LIN {X 0,Y 421.046,Z 301.335,A -85,B 0,C 180,E1 -10144.338,E2 -10144.338} C_VEL
LIN {X 0,Y 421.385,Z 304.023,A -85,B 0,C 180,E1 -10144.837,E2 -10144.837} C_VEL
LIN {X 0,Y 420.511,Z 320.205,A -85,B 0,C 180,E1 -10147.657,E2 -10147.657} C_VEL
LIN {X 0,Y 419.69,Z 337.101,A -85,B 0,C 180,E1 -10150.579,E2 -10150.579} C_VEL
LIN {X 0,Y 422.949,Z 357.604,A -85,B 0,C 180,E1 -10151.184,E2 -10151.184} C_VEL
LIN {X 0,Y 424.065,Z 368.601,A -85,B 0,C 180,E1 -10151.466,E2 -10151.466} C_VEL
LIN {X 0,Y 422.703,Z 448.202,A -85,B 0,C 180,E1 -10153.026,E2 -10153.026} C_VEL
LIN {X 0,Y 422.076,Z 462.168,A -85,B 0,C 180,E1 -10153.498,E2 -10153.498} C_VEL
LIN {X 0,Y 421.349,Z 475.179,A -85,B 0,C 180,E1 -10154.153,E2 -10154.153} C_VEL
LIN {X 0,Y 420.586,Z 487.585,A -85,B 0,C 180,E1 -10154.992,E2 -10154.992} C_VEL
LIN {X 0,Y 419.764,Z 499.223,A -85,B 0,C 180,E1 -10156.002,E2 -10156.002} C_VEL
LIN {X 0,Y 419.009,Z 509.823,A -85,B 0,C 180,E1 -10157.162,E2 -10157.162} C_VEL
LIN {X 0,Y 418.449,Z 518.856,A -85,B 0,C 180,E1 -10158.375,E2 -10158.375} C_VEL
LIN {X 0,Y 417.83,Z 527.672,A -85,B 0,C 180,E1 -10159.83,E2 -10159.83} C_VEL
LIN {X 0,Y 417.483,Z 534.743,A -85,B 0,C 180,E1 -10161.288,E2 -10161.288} C_VEL
LIN {X 0,Y 417.25,Z 540.419,A -85,B 0,C 180,E1 -10162.745,E2 -10162.745} C_VEL
LIN {X 0,Y 417.115,Z 544.874,A -85,B 0,C 180,E1 -10164.2,E2 -10164.2} C_VEL
LIN {X 0,Y 417.146,Z 547.246,A -85,B 0,C 180,E1 -10165.17,E2 -10165.17} C_VEL
LIN {X 0,Y 417.051,Z 549.135,A -85,B 0,C 180,E1 -10166.137,E2 -10166.137} C_VEL
LIN {X 0,Y 417.124,Z 550.576,A -85,B 0,C 180,E1 -10167.105,E2 -10167.105} C_VEL
LIN {X 0,Y 417.122,Z 551.604,A -85,B 0,C 180,E1 -10168.071,E2 -10168.071} C_VEL
LIN {X 0,Y 417.096,Z 552.225,A -85,B 0,C 180,E1 -10169.036,E2 -10169.036} C_VEL
LIN {X 0,Y 417.123,Z 552.395,A -85,B 0,C 180,E1 -10170.002,E2 -10170.002} C_VEL
LIN {X 0,Y 417.109,Z 552.146,A -85,B 0,C 180,E1 -10170.967,E2 -10170.967} C_VEL
LIN {X 0,Y 417.123,Z 551.496,A -85,B 0,C 180,E1 -10171.932,E2 -10171.932} C_VEL
LIN {X 0,Y 417.156,Z 550.435,A -85,B 0,C 180,E1 -10172.898,E2 -10172.898} C_VEL
LIN {X 0,Y 417.054,Z 548.89,A -85,B 0,C 180,E1 -10173.866,E2 -10173.866} C_VEL
LIN {X 0,Y 417.143,Z 545.765,A -85,B 0,C 180,E1 -10175.318,E2 -10175.318} C_VEL
LIN {X 0,Y 417.233,Z 541.533,A -85,B 0,C 180,E1 -10176.772,E2 -10176.772} C_VEL
LIN {X 0,Y 417.443,Z 535.054,A -85,B 0,C 180,E1 -10178.472,E2 -10178.472} C_VEL
LIN {X 0,Y 417.739,Z 527.969,A -85,B 0,C 180,E1 -10179.931,E2 -10179.931} C_VEL
LIN {X 0,Y 418.276,Z 519.076,A -85,B 0,C 180,E1 -10181.387,E2 -10181.387} C_VEL
LIN {X 0,Y 418.823,Z 509.96,A -85,B 0,C 180,E1 -10182.6,E2 -10182.6} C_VEL
LIN {X 0,Y 419.403,Z 499.932,A -85,B 0,C 180,E1 -10183.692,E2 -10183.692} C_VEL
LIN {X 0,Y 420.108,Z 488.819,A -85,B 0,C 180,E1 -10184.657,E2 -10184.657} C_VEL
LIN {X 0,Y 420.808,Z 476.413,A -85,B 0,C 180,E1 -10185.499,E2 -10185.499} C_VEL
LIN {X 0,Y 421.393,Z 464.719,A -85,B 0,C 180,E1 -10186.097,E2 -10186.097} C_VEL
LIN {X 0,Y 421.903,Z 452.292,A -85,B 0,C 180,E1 -10186.543,E2 -10186.543} C_VEL
LIN {X 0,Y 422.237,Z 433.946,A -85,B 0,C 180,E1 -10186.935,E2 -10186.935} C_VEL
LIN {X 0,Y 423.043,Z 365.545,A -85,B 0,C 180,E1 -10188.216,E2 -10188.216} C_VEL
LIN {X 0,Y 419.504,Z 339.754,A -85,B 0,C 180,E1 -10188.877,E2 -10188.877} C_VEL
LIN {X 0,Y 420.603,Z 320.904,A -85,B 0,C 180,E1 -10192.341,E2 -10192.341} C_VEL
LIN {X 0,Y 421.565,Z 304.734,A -85,B 0,C 180,E1 -10195.354,E2 -10195.354} C_VEL
LIN {X 0,Y 418.666,Z 290.263,A -85,B 0,C 180,E1 -10198.307,E2 -10198.307} C_VEL
LIN {X 0,Y 418.272,Z 288.385,A -85,B 0,C 180,E1 -10198.733,E2 -10198.733} C_VEL
LIN {X 0,Y 418.205,Z 288.39,A -85,B 0,C 180,E1 -10201.395,E2 -10201.395} C_VEL
LIN {X 0,Y 418.246,Z 288.389,A -85,B 0,C 180,E1 -10204.576,E2 -10204.576} C_VEL
LIN {X 0,Y 418.209,Z 288.388,A -85,B 0,C 180,E1 -10207.829,E2 -10207.829} C_VEL
LIN {X 0,Y 418.197,Z 288.393,A -85,B 0,C 180,E1 -10210.948,E2 -10210.948} C_VEL
LIN {X 0,Y 418.19,Z 288.39,A -85,B 0,C 180,E1 -10213.726,E2 -10213.726} C_VEL
LIN {X 0,Y 418.186,Z 288.393,A -85,B 0,C 180,E1 -10216.445,E2 -10216.445} C_VEL
LIN {X 0,Y 418.192,Z 288.393,A -85,B 0,C 180,E1 -10219.131,E2 -10219.131} C_VEL
LIN {X 0,Y 418.217,Z 288.393,A -85,B 0,C 180,E1 -10222.773,E2 -10222.773} C_VEL
LIN {X 0,Y 418.211,Z 288.389,A -85,B 0,C 180,E1 -10226.319,E2 -10226.319} C_VEL
LIN {X 0,Y 418.22,Z 288.388,A -85,B 0,C 180,E1 -10229.725,E2 -10229.725} C_VEL
LIN {X 0,Y 418.239,Z 288.389,A -85,B 0,C 180,E1 -10233.018,E2 -10233.018} C_VEL
LIN {X 0,Y 418.24,Z 288.385,A -85,B 0,C 180,E1 -10236.216,E2 -10236.216} C_VEL
LIN {X 0,Y 418.22,Z 288.389,A -85,B 0,C 180,E1 -10239.335,E2 -10239.335} C_VEL
LIN {X 0,Y 418.249,Z 288.384,A -85,B 0,C 180,E1 -10242.394,E2 -10242.394} C_VEL
LIN {X 0,Y 418.27,Z 288.383,A -85,B 0,C 180,E1 -10245.401,E2 -10245.401} C_VEL
LIN {X 0,Y 418.291,Z 288.379,A -85,B 0,C 180,E1 -10248.368,E2 -10248.368} C_VEL
LIN {X 0,Y 418.484,Z 288.355,A -85,B 0,C 180,E1 -10252.278,E2 -10252.278} C_VEL
LIN {X 0,Y 418.474,Z 288.357,A -85,B 0,C 180,E1 -10254.216,E2 -10254.216} C_VEL
LIN {X 0,Y 418.508,Z 288.354,A -85,B 0,C 180,E1 -10258.075,E2 -10258.075} C_VEL
LIN {X 0,Y 418.636,Z 288.337,A -85,B 0,C 180,E1 -10260,E2 -10260} C_VEL
LIN {X 0,Y 418.466,Z 288.359,A -85,B 0,C 180,E1 -10262.888,E2 -10262.888} C_VEL
LIN {X 0,Y 418.456,Z 288.36,A -85,B 0,C 180,E1 -10266.751,E2 -10266.751} C_VEL
LIN {X 0,Y 418.313,Z 288.378,A -85,B 0,C 180,E1 -10269.672,E2 -10269.672} C_VEL
LIN {X 0,Y 418.325,Z 288.377,A -85,B 0,C 180,E1 -10273.006,E2 -10273.006} C_VEL
LIN {X 0,Y 418.282,Z 288.381,A -85,B 0,C 180,E1 -10276.735,E2 -10276.735} C_VEL
LIN {X 0,Y 418.24,Z 288.387,A -85,B 0,C 180,E1 -10279.79,E2 -10279.79} C_VEL
LIN {X 0,Y 418.21,Z 288.39,A -85,B 0,C 180,E1 -10282.737,E2 -10282.737} C_VEL
LIN {X 0,Y 418.243,Z 288.386,A -85,B 0,C 180,E1 -10285.905,E2 -10285.905} C_VEL
LIN {X 0,Y 418.248,Z 288.386,A -85,B 0,C 180,E1 -10289.163,E2 -10289.163} C_VEL
LIN {X 0,Y 418.234,Z 288.387,A -85,B 0,C 180,E1 -10292.845,E2 -10292.845} C_VEL
LIN {X 0,Y 418.226,Z 288.389,A -85,B 0,C 180,E1 -10296.24,E2 -10296.24} C_VEL
LIN {X 0,Y 418.245,Z 288.387,A -85,B 0,C 180,E1 -10299.682,E2 -10299.682} C_VEL
LIN {X 0,Y 418.227,Z 288.39,A -85,B 0,C 180,E1 -10302.325,E2 -10302.325} C_VEL
LIN {X 0,Y 418.233,Z 288.387,A -85,B 0,C 180,E1 -10305.112,E2 -10305.112} C_VEL
LIN {X 0,Y 418.277,Z 288.382,A -85,B 0,C 180,E1 -10307.775,E2 -10307.775} C_VEL
LIN {X 0,Y 418.254,Z 288.386,A -85,B 0,C 180,E1 -10311.561,E2 -10311.561} C_VEL
LIN {X 0,Y 418.249,Z 288.385,A -85,B 0,C 180,E1 -10315.16,E2 -10315.16} C_VEL
LIN {X 0,Y 418.235,Z 288.387,A -85,B 0,C 180,E1 -10317.473,E2 -10317.473} C_VEL
LIN {X 0,Y 418.261,Z 288.385,A -85,B 0,C 180,E1 -10320.896,E2 -10320.896} C_VEL
LIN {X 0,Y 418.264,Z 288.384,A -85,B 0,C 180,E1 -10324.097,E2 -10324.097} C_VEL
LIN {X 0,Y 418.233,Z 288.387,A -85,B 0,C 180,E1 -10327.264,E2 -10327.264} C_VEL
LIN {X 0,Y 418.279,Z 288.382,A -85,B 0,C 180,E1 -10330.364,E2 -10330.364} C_VEL
LIN {X 0,Y 418.314,Z 288.377,A -85,B 0,C 180,E1 -10333.405,E2 -10333.405} C_VEL
LIN {X 0,Y 418.343,Z 288.375,A -85,B 0,C 180,E1 -10336.999,E2 -10336.999} C_VEL
LIN {X 0,Y 418.339,Z 288.374,A -85,B 0,C 180,E1 -10340.328,E2 -10340.328} C_VEL
LIN {X 0,Y 418.511,Z 288.353,A -85,B 0,C 180,E1 -10342.279,E2 -10342.279} C_VEL
LIN {X 0,Y 418.511,Z 288.352,A -85,B 0,C 180,E1 -10344.216,E2 -10344.216} C_VEL
LIN {X 0,Y 418.542,Z 288.348,A -85,B 0,C 180,E1 -10348.074,E2 -10348.074} C_VEL
LIN {X 0,Y 418.67,Z 288.332,A -85,B 0,C 180,E1 -10349.998,E2 -10349.998} C_VEL
LIN {X 0,Y 418.507,Z 288.357,A -85,B 0,C 180,E1 -10352.886,E2 -10352.886} C_VEL
LIN {X 0,Y 418.482,Z 288.358,A -85,B 0,C 180,E1 -10356.749,E2 -10356.749} C_VEL
LIN {X 0,Y 418.352,Z 288.371,A -85,B 0,C 180,E1 -10359.17,E2 -10359.17} C_VEL
LIN {X 0,Y 418.363,Z 288.371,A -85,B 0,C 180,E1 -10362.611,E2 -10362.611} C_VEL
LIN {X 0,Y 418.324,Z 288.376,A -85,B 0,C 180,E1 -10363.36,E2 -10363.36} C_VEL
LIN {X 0,Y 417.633,Z 288.461,A -85,B 0,C 180,E1 -10364.163,E2 -10364.163} C_VEL
LIN {X 0,Y 414.749,Z 288.82,A -85,B 0,C 180,E1 -10365.468,E2 -10365.468} C_VEL
LIN {X 0,Y 412.33,Z 289.122,A -85,B 0,C 180,E1 -10366.522,E2 -10366.522} C_VEL
LIN {X 0,Y 411.306,Z 289.25,A -85,B 0,C 180,E1 -10367.337,E2 -10367.337} C_VEL
LIN {X 0,Y 411.23,Z 289.257,A -85,B 0,C 180,E1 -10367.613,E2 -10367.613} C_VEL
LIN {X 0,Y 411.221,Z 289.265,A -85,B 0,C 180,E1 -10371.029,E2 -10371.029} C_VEL
LIN {X 0,Y 411.214,Z 289.26,A -85,B 0,C 180,E1 -10374.212,E2 -10374.212} C_VEL
LIN {X 0,Y 411.243,Z 289.258,A -85,B 0,C 180,E1 -10377.474,E2 -10377.474} C_VEL
LIN {X 0,Y 411.182,Z 289.266,A -85,B 0,C 180,E1 -10380.843,E2 -10380.843} C_VEL
LIN {X 0,Y 411.183,Z 289.263,A -85,B 0,C 180,E1 -10384.33,E2 -10384.33} C_VEL
LIN {X 0,Y 411.179,Z 289.264,A -85,B 0,C 180,E1 -10387.969,E2 -10387.969} C_VEL
LIN {X 0,Y 411.255,Z 289.359,A -85,B 0,C 180,E1 -10391.508,E2 -10391.508} C_VEL
LIN {X 0,Y 412.397,Z 295.233,A -85,B 0,C 180,E1 -10392.933,E2 -10392.933} C_VEL
LIN {X 0,Y 414.802,Z 304.457,A -85,B 0,C 180,E1 -10393.227,E2 -10393.227} C_VEL
LIN {X 0,Y 416.781,Z 315.123,A -85,B 0,C 180,E1 -10393.524,E2 -10393.524} C_VEL
LIN {X 0,Y 415.341,Z 403.223,A -85,B 0,C 180,E1 -10395.224,E2 -10395.224} C_VEL
LIN {X 0,Y 415.04,Z 416.613,A -85,B 0,C 180,E1 -10395.683,E2 -10395.683} C_VEL
LIN {X 0,Y 414.55,Z 428.862,A -85,B 0,C 180,E1 -10396.29,E2 -10396.29} C_VEL
LIN {X 0,Y 413.945,Z 441.31,A -85,B 0,C 180,E1 -10397.127,E2 -10397.127} C_VEL
LIN {X 0,Y 413.301,Z 452.924,A -85,B 0,C 180,E1 -10398.132,E2 -10398.132} C_VEL
LIN {X 0,Y 412.687,Z 462.758,A -85,B 0,C 180,E1 -10399.193,E2 -10399.193} C_VEL
LIN {X 0,Y 412.002,Z 473.088,A -85,B 0,C 180,E1 -10400.583,E2 -10400.583} C_VEL
LIN {X 0,Y 411.43,Z 481.862,A -85,B 0,C 180,E1 -10402.053,E2 -10402.053} C_VEL
LIN {X 0,Y 410.983,Z 488.662,A -85,B 0,C 180,E1 -10403.476,E2 -10403.476} C_VEL
LIN {X 0,Y 410.578,Z 495.276,A -85,B 0,C 180,E1 -10405.237,E2 -10405.237} C_VEL
LIN {X 0,Y 410.367,Z 499.644,A -85,B 0,C 180,E1 -10406.768,E2 -10406.768} C_VEL
LIN {X 0,Y 410.18,Z 502.139,A -85,B 0,C 180,E1 -10407.917,E2 -10407.917} C_VEL
LIN {X 0,Y 410.024,Z 504.05,A -85,B 0,C 180,E1 -10409.056,E2 -10409.056} C_VEL
LIN {X 0,Y 409.943,Z 505.913,A -85,B 0,C 180,E1 -10410.953,E2 -10410.953} C_VEL
LIN {X 0,Y 409.95,Z 506.241,A -85,B 0,C 180,E1 -10413.043,E2 -10413.043} C_VEL
LIN {X 0,Y 410.043,Z 505.234,A -85,B 0,C 180,E1 -10414.629,E2 -10414.629} C_VEL
LIN {X 0,Y 410.195,Z 503.889,A -85,B 0,C 180,E1 -10415.72,E2 -10415.72} C_VEL
LIN {X 0,Y 410.366,Z 502.082,A -85,B 0,C 180,E1 -10416.803,E2 -10416.803} C_VEL
LIN {X 0,Y 410.635,Z 498.359,A -85,B 0,C 180,E1 -10418.41,E2 -10418.41} C_VEL
LIN {X 0,Y 411.045,Z 493.008,A -85,B 0,C 180,E1 -10420.095,E2 -10420.095} C_VEL
LIN {X 0,Y 411.519,Z 486.934,A -85,B 0,C 180,E1 -10421.583,E2 -10421.583} C_VEL
LIN {X 0,Y 412.174,Z 478.896,A -85,B 0,C 180,E1 -10423.15,E2 -10423.15} C_VEL
LIN {X 0,Y 412.849,Z 470.57,A -85,B 0,C 180,E1 -10424.448,E2 -10424.448} C_VEL
LIN {X 0,Y 413.65,Z 460.35,A -85,B 0,C 180,E1 -10425.74,E2 -10425.74} C_VEL
LIN {X 0,Y 414.424,Z 450.265,A -85,B 0,C 180,E1 -10426.766,E2 -10426.766} C_VEL
LIN {X 0,Y 415.041,Z 439.361,A -85,B 0,C 180,E1 -10427.656,E2 -10427.656} C_VEL
LIN {X 0,Y 415.674,Z 427.031,A -85,B 0,C 180,E1 -10428.435,E2 -10428.435} C_VEL
LIN {X 0,Y 416.13,Z 414.173,A -85,B 0,C 180,E1 -10429.032,E2 -10429.032} C_VEL
LIN {X 0,Y 416.469,Z 401.016,A -85,B 0,C 180,E1 -10429.426,E2 -10429.426} C_VEL
LIN {X 0,Y 418.135,Z 314.185,A -85,B 0,C 180,E1 -10431.159,E2 -10431.159} C_VEL
LIN {X 0,Y 415.58,Z 302.673,A -85,B 0,C 180,E1 -10431.56,E2 -10431.56} C_VEL
LIN {X 0,Y 412.825,Z 295.614,A -85,B 0,C 180,E1 -10431.896,E2 -10431.896} C_VEL
LIN {X 0,Y 411.408,Z 289.242,A -85,B 0,C 180,E1 -10433.194,E2 -10433.194} C_VEL
LIN {X 0,Y 411.417,Z 289.242,A -85,B 0,C 180,E1 -10437.063,E2 -10437.063} C_VEL
LIN {X 0,Y 411.586,Z 289.215,A -85,B 0,C 180,E1 -10440,E2 -10440} C_VEL
LIN {X 0,Y 411.417,Z 289.238,A -85,B 0,C 180,E1 -10442.938,E2 -10442.938} C_VEL
LIN {X 0,Y 411.404,Z 289.24,A -85,B 0,C 180,E1 -10446.868,E2 -10446.868} C_VEL
LIN {X 0,Y 411.246,Z 289.256,A -85,B 0,C 180,E1 -10449.84,E2 -10449.84} C_VEL
LIN {X 0,Y 411.264,Z 289.256,A -85,B 0,C 180,E1 -10453.11,E2 -10453.11} C_VEL
LIN {X 0,Y 411.21,Z 289.264,A -85,B 0,C 180,E1 -10456.891,E2 -10456.891} C_VEL
LIN {X 0,Y 411.163,Z 289.263,A -85,B 0,C 180,E1 -10459.991,E2 -10459.991} C_VEL
LIN {X 0,Y 411.157,Z 289.267,A -85,B 0,C 180,E1 -10463.151,E2 -10463.151} C_VEL
LIN {X 0,Y 411.195,Z 289.259,A -85,B 0,C 180,E1 -10466.384,E2 -10466.384} C_VEL
LIN {X 0,Y 411.16,Z 289.268,A -85,B 0,C 180,E1 -10469.716,E2 -10469.716} C_VEL
LIN {X 0,Y 411.169,Z 289.271,A -85,B 0,C 180,E1 -10473.16,E2 -10473.16} C_VEL
LIN {X 0,Y 411.16,Z 289.267,A -85,B 0,C 180,E1 -10476.557,E2 -10476.557} C_VEL
LIN {X 0,Y 411.195,Z 289.262,A -85,B 0,C 180,E1 -10479.734,E2 -10479.734} C_VEL
LIN {X 0,Y 411.148,Z 289.271,A -85,B 0,C 180,E1 -10483.137,E2 -10483.137} C_VEL
LIN {X 0,Y 411.141,Z 289.27,A -85,B 0,C 180,E1 -10485.886,E2 -10485.886} C_VEL
LIN {X 0,Y 411.139,Z 289.271,A -85,B 0,C 180,E1 -10488.776,E2 -10488.776} C_VEL
LIN {X 0,Y 411.168,Z 289.267,A -85,B 0,C 180,E1 -10492.03,E2 -10492.03} C_VEL
LIN {X 0,Y 411.188,Z 289.272,A -85,B 0,C 180,E1 -10495.671,E2 -10495.671} C_VEL
LIN {X 0,Y 411.174,Z 289.277,A -85,B 0,C 180,E1 -10499.156,E2 -10499.156} C_VEL
LIN {X 0,Y 411.242,Z 289.392,A -85,B 0,C 180,E1 -10501.493,E2 -10501.493} C_VEL
LIN {X 0,Y 414.104,Z 302.418,A -85,B 0,C 180,E1 -10504.092,E2 -10504.092} C_VEL
LIN {X 0,Y 414.521,Z 305.674,A -85,B 0,C 180,E1 -10504.715,E2 -10504.715} C_VEL
LIN {X 0,Y 413.497,Z 322.95,A -85,B 0,C 180,E1 -10507.784,E2 -10507.784} C_VEL
LIN {X 0,Y 412.843,Z 336.588,A -85,B 0,C 180,E1 -10510.177,E2 -10510.177} C_VEL
LIN {X 0,Y 416.359,Z 358.576,A -85,B 0,C 180,E1 -10510.855,E2 -10510.855} C_VEL
LIN {X 0,Y 417.425,Z 369.282,A -85,B 0,C 180,E1 -10511.137,E2 -10511.137} C_VEL
LIN {X 0,Y 415.99,Z 447.96,A -85,B 0,C 180,E1 -10512.712,E2 -10512.712} C_VEL
LIN {X 0,Y 415.37,Z 461.098,A -85,B 0,C 180,E1 -10513.16,E2 -10513.16} C_VEL
LIN {X 0,Y 414.685,Z 473.298,A -85,B 0,C 180,E1 -10513.765,E2 -10513.765} C_VEL
LIN {X 0,Y 413.791,Z 485.957,A -85,B 0,C 180,E1 -10514.614,E2 -10514.614} C_VEL
LIN {X 0,Y 412.985,Z 497.705,A -85,B 0,C 180,E1 -10515.629,E2 -10515.629} C_VEL
LIN {X 0,Y 412.225,Z 507.992,A -85,B 0,C 180,E1 -10516.746,E2 -10516.746} C_VEL
LIN {X 0,Y 411.465,Z 518.593,A -85,B 0,C 180,E1 -10518.175,E2 -10518.175} C_VEL
LIN {X 0,Y 410.8,Z 527.377,A -85,B 0,C 180,E1 -10519.654,E2 -10519.654} C_VEL
LIN {X 0,Y 410.427,Z 534.434,A -85,B 0,C 180,E1 -10521.137,E2 -10521.137} C_VEL
LIN {X 0,Y 410.17,Z 540.096,A -85,B 0,C 180,E1 -10522.619,E2 -10522.619} C_VEL
LIN {X 0,Y 410.036,Z 544.536,A -85,B 0,C 180,E1 -10524.099,E2 -10524.099} C_VEL
LIN {X 0,Y 410.053,Z 546.905,A -85,B 0,C 180,E1 -10525.086,E2 -10525.086} C_VEL
LIN {X 0,Y 409.968,Z 548.774,A -85,B 0,C 180,E1 -10526.07,E2 -10526.07} C_VEL
LIN {X 0,Y 410.022,Z 550.205,A -85,B 0,C 180,E1 -10527.054,E2 -10527.054} C_VEL
LIN {X 0,Y 410.048,Z 551.226,A -85,B 0,C 180,E1 -10528.037,E2 -10528.037} C_VEL
LIN {X 0,Y 410.016,Z 551.834,A -85,B 0,C 180,E1 -10529.02,E2 -10529.02} C_VEL
LIN {X 0,Y 410.039,Z 551.988,A -85,B 0,C 180,E1 -10530.002,E2 -10530.002} C_VEL
LIN {X 0,Y 410.028,Z 551.73,A -85,B 0,C 180,E1 -10530.984,E2 -10530.984} C_VEL
LIN {X 0,Y 410.051,Z 551.071,A -85,B 0,C 180,E1 -10531.966,E2 -10531.966} C_VEL
LIN {X 0,Y 410.054,Z 549.99,A -85,B 0,C 180,E1 -10532.949,E2 -10532.949} C_VEL
LIN {X 0,Y 409.97,Z 548.429,A -85,B 0,C 180,E1 -10533.933,E2 -10533.933} C_VEL
LIN {X 0,Y 410.059,Z 545.275,A -85,B 0,C 180,E1 -10535.41,E2 -10535.41} C_VEL
LIN {X 0,Y 410.165,Z 541.011,A -85,B 0,C 180,E1 -10536.89,E2 -10536.89} C_VEL
LIN {X 0,Y 410.363,Z 534.489,A -85,B 0,C 180,E1 -10538.619,E2 -10538.619} C_VEL
LIN {X 0,Y 410.693,Z 527.341,A -85,B 0,C 180,E1 -10540.103,E2 -10540.103} C_VEL
LIN {X 0,Y 411.273,Z 518.382,A -85,B 0,C 180,E1 -10541.583,E2 -10541.583} C_VEL
LIN {X 0,Y 411.876,Z 509.197,A -85,B 0,C 180,E1 -10542.816,E2 -10542.816} C_VEL
LIN {X 0,Y 412.474,Z 499.048,A -85,B 0,C 180,E1 -10543.926,E2 -10543.926} C_VEL
LIN {X 0,Y 413.198,Z 487.791,A -85,B 0,C 180,E1 -10544.907,E2 -10544.907} C_VEL
LIN {X 0,Y 413.941,Z 475.22,A -85,B 0,C 180,E1 -10545.763,E2 -10545.763} C_VEL
LIN {X 0,Y 414.535,Z 463.156,A -85,B 0,C 180,E1 -10546.371,E2 -10546.371} C_VEL
LIN {X 0,Y 415.081,Z 449.036,A -85,B 0,C 180,E1 -10546.855,E2 -10546.855} C_VEL
LIN {X 0,Y 415.934,Z 395.669,A -85,B 0,C 180,E1 -10547.89,E2 -10547.89} C_VEL
LIN {X 0,Y 416.24,Z 366.622,A -85,B 0,C 180,E1 -10548.454,E2 -10548.454} C_VEL
LIN {X 0,Y 412.547,Z 339.36,A -85,B 0,C 180,E1 -10549.175,E2 -10549.175} C_VEL
LIN {X 0,Y 413.717,Z 320.343,A -85,B 0,C 180,E1 -10552.734,E2 -10552.734} C_VEL
LIN {X 0,Y 414.634,Z 306.778,A -85,B 0,C 180,E1 -10555.305,E2 -10555.305} C_VEL
LIN {X 0,Y 412.16,Z 293.628,A -85,B 0,C 180,E1 -10558.014,E2 -10558.014} C_VEL
LIN {X 0,Y 411.234,Z 289.261,A -85,B 0,C 180,E1 -10558.948,E2 -10558.948} C_VEL
LIN {X 0,Y 411.159,Z 289.269,A -85,B 0,C 180,E1 -10561.996,E2 -10561.996} C_VEL
LIN {X 0,Y 411.196,Z 289.266,A -85,B 0,C 180,E1 -10564.875,E2 -10564.875} C_VEL
LIN {X 0,Y 411.183,Z 289.264,A -85,B 0,C 180,E1 -10568.164,E2 -10568.164} C_VEL
LIN {X 0,Y 411.15,Z 289.267,A -85,B 0,C 180,E1 -10571.806,E2 -10571.806} C_VEL
LIN {X 0,Y 411.16,Z 289.267,A -85,B 0,C 180,E1 -10575.507,E2 -10575.507} C_VEL
LIN {X 0,Y 411.133,Z 289.275,A -85,B 0,C 180,E1 -10578.772,E2 -10578.772} C_VEL
LIN {X 0,Y 411.166,Z 289.266,A -85,B 0,C 180,E1 -10582.023,E2 -10582.023} C_VEL
LIN {X 0,Y 411.183,Z 289.267,A -85,B 0,C 180,E1 -10585.122,E2 -10585.122} C_VEL
LIN {X 0,Y 411.14,Z 289.269,A -85,B 0,C 180,E1 -10588,E2 -10588} C_VEL
LIN {X 0,Y 411.191,Z 289.264,A -85,B 0,C 180,E1 -10591.407,E2 -10591.407} C_VEL
LIN {X 0,Y 411.19,Z 289.268,A -85,B 0,C 180,E1 -10594.932,E2 -10594.932} C_VEL
LIN {X 0,Y 411.176,Z 289.266,A -85,B 0,C 180,E1 -10597.911,E2 -10597.911} C_VEL
LIN {X 0,Y 411.19,Z 289.268,A -85,B 0,C 180,E1 -10601.049,E2 -10601.049} C_VEL
LIN {X 0,Y 411.226,Z 289.259,A -85,B 0,C 180,E1 -10604.13,E2 -10604.13} C_VEL
LIN {X 0,Y 411.275,Z 289.257,A -85,B 0,C 180,E1 -10607.164,E2 -10607.164} C_VEL
LIN {X 0,Y 411.264,Z 289.255,A -85,B 0,C 180,E1 -10610.16,E2 -10610.16} C_VEL
LIN {X 0,Y 411.425,Z 289.239,A -85,B 0,C 180,E1 -10613.132,E2 -10613.132} C_VEL
LIN {X 0,Y 411.273,Z 289.257,A -85,B 0,C 180,E1 -10615.098,E2 -10615.098} C_VEL
LIN {X 0,Y 411.477,Z 289.229,A -85,B 0,C 180,E1 -10618.042,E2 -10618.042} C_VEL
LIN {X 0,Y 411.606,Z 289.213,A -85,B 0,C 180,E1 -10620,E2 -10620} C_VEL
LIN {X 0,Y 411.423,Z 289.237,A -85,B 0,C 180,E1 -10622.937,E2 -10622.937} C_VEL
LIN {X 0,Y 411.42,Z 289.236,A -85,B 0,C 180,E1 -10626.867,E2 -10626.867} C_VEL
LIN {X 0,Y 411.266,Z 289.256,A -85,B 0,C 180,E1 -10629.839,E2 -10629.839} C_VEL
LIN {X 0,Y 411.283,Z 289.254,A -85,B 0,C 180,E1 -10633.108,E2 -10633.108} C_VEL
LIN {X 0,Y 411.229,Z 289.26,A -85,B 0,C 180,E1 -10636.889,E2 -10636.889} C_VEL
LIN {X 0,Y 411.182,Z 289.266,A -85,B 0,C 180,E1 -10639.989,E2 -10639.989} C_VEL
LIN {X 0,Y 411.175,Z 289.267,A -85,B 0,C 180,E1 -10643.149,E2 -10643.149} C_VEL
LIN {X 0,Y 411.212,Z 289.263,A -85,B 0,C 180,E1 -10646.382,E2 -10646.382} C_VEL
LIN {X 0,Y 411.185,Z 289.266,A -85,B 0,C 180,E1 -10649.713,E2 -10649.713} C_VEL
LIN {X 0,Y 411.184,Z 289.266,A -85,B 0,C 180,E1 -10653.157,E2 -10653.157} C_VEL
LIN {X 0,Y 411.174,Z 289.268,A -85,B 0,C 180,E1 -10656.554,E2 -10656.554} C_VEL
LIN {X 0,Y 411.208,Z 289.263,A -85,B 0,C 180,E1 -10659.731,E2 -10659.731} C_VEL
LIN {X 0,Y 411.16,Z 289.268,A -85,B 0,C 180,E1 -10663.135,E2 -10663.135} C_VEL
LIN {X 0,Y 411.205,Z 289.263,A -85,B 0,C 180,E1 -10665.875,E2 -10665.875} C_VEL
LIN {X 0,Y 411.196,Z 289.265,A -85,B 0,C 180,E1 -10668.766,E2 -10668.766} C_VEL
LIN {X 0,Y 411.192,Z 289.265,A -85,B 0,C 180,E1 -10672.029,E2 -10672.029} C_VEL
LIN {X 0,Y 411.196,Z 289.265,A -85,B 0,C 180,E1 -10675.668,E2 -10675.668} C_VEL
LIN {X 0,Y 411.18,Z 289.265,A -85,B 0,C 180,E1 -10679.153,E2 -10679.153} C_VEL
LIN {X 0,Y 411.252,Z 289.259,A -85,B 0,C 180,E1 -10682.523,E2 -10682.523} C_VEL
LIN {X 0,Y 411.221,Z 289.261,A -85,B 0,C 180,E1 -10685.785,E2 -10685.785} C_VEL
LIN {X 0,Y 411.192,Z 289.265,A -85,B 0,C 180,E1 -10688.966,E2 -10688.966} C_VEL
LIN {X 0,Y 411.249,Z 289.257,A -85,B 0,C 180,E1 -10692.085,E2 -10692.085} C_VEL
LIN {X 0,Y 411.257,Z 289.256,A -85,B 0,C 180,E1 -10695.147,E2 -10695.147} C_VEL
LIN {X 0,Y 411.281,Z 289.253,A -85,B 0,C 180,E1 -10698.167,E2 -10698.167} C_VEL
LIN {X 0,Y 411.48,Z 289.228,A -85,B 0,C 180,E1 -10702.146,E2 -10702.146} C_VEL
LIN {X 0,Y 411.473,Z 289.229,A -85,B 0,C 180,E1 -10704.117,E2 -10704.117} C_VEL
LIN {X 0,Y 411.511,Z 289.224,A -85,B 0,C 180,E1 -10708.041,E2 -10708.041} C_VEL
LIN {X 0,Y 411.639,Z 289.208,A -85,B 0,C 180,E1 -10709.998,E2 -10709.998} C_VEL
LIN {X 0,Y 411.463,Z 289.234,A -85,B 0,C 180,E1 -10712.935,E2 -10712.935} C_VEL
LIN {X 0,Y 411.45,Z 289.236,A -85,B 0,C 180,E1 -10716.865,E2 -10716.865} C_VEL
LIN {X 0,Y 411.349,Z 289.248,A -85,B 0,C 180,E1 -10718.843,E2 -10718.843} C_VEL
LIN {X 0,Y 411.292,Z 289.25,A -85,B 0,C 180,E1 -10721.83,E2 -10721.83} C_VEL
LIN {X 0,Y 411.254,Z 289.259,A -85,B 0,C 180,E1 -10724.85,E2 -10724.85} C_VEL
LIN {X 0,Y 411.23,Z 289.257,A -85,B 0,C 180,E1 -10727.613,E2 -10727.613} C_VEL
LIN {X 0,Y 410.579,Z 289.341,A -85,B 0,C 180,E1 -10728.431,E2 -10728.431} C_VEL
LIN {X 0,Y 407.715,Z 289.696,A -85,B 0,C 180,E1 -10729.76,E2 -10729.76} C_VEL
LIN {X 0,Y 405.283,Z 290.002,A -85,B 0,C 180,E1 -10730.833,E2 -10730.833} C_VEL
LIN {X 0,Y 404.241,Z 290.128,A -85,B 0,C 180,E1 -10731.663,E2 -10731.663} C_VEL
LIN {X 0,Y 404.159,Z 290.138,A -85,B 0,C 180,E1 -10731.944,E2 -10731.944} C_VEL
LIN {X 0,Y 404.201,Z 290.136,A -85,B 0,C 180,E1 -10735.293,E2 -10735.293} C_VEL
LIN {X 0,Y 404.181,Z 290.135,A -85,B 0,C 180,E1 -10737.996,E2 -10737.996} C_VEL
LIN {X 0,Y 404.127,Z 290.144,A -85,B 0,C 180,E1 -10741.556,E2 -10741.556} C_VEL
LIN {X 0,Y 404.162,Z 290.142,A -85,B 0,C 180,E1 -10745.012,E2 -10745.012} C_VEL
LIN {X 0,Y 404.138,Z 290.142,A -85,B 0,C 180,E1 -10748.752,E2 -10748.752} C_VEL
LIN {X 0,Y 404.192,Z 290.207,A -85,B 0,C 180,E1 -10751.307,E2 -10751.307} C_VEL
LIN {X 0,Y 405.304,Z 295.784,A -85,B 0,C 180,E1 -10752.642,E2 -10752.642} C_VEL
LIN {X 0,Y 407.678,Z 303.954,A -85,B 0,C 180,E1 -10752.914,E2 -10752.914} C_VEL
LIN {X 0,Y 409.938,Z 315.032,A -85,B 0,C 180,E1 -10753.239,E2 -10753.239} C_VEL
LIN {X 0,Y 408.487,Z 403.598,A -85,B 0,C 180,E1 -10754.986,E2 -10754.986} C_VEL
LIN {X 0,Y 408.133,Z 416.613,A -85,B 0,C 180,E1 -10755.436,E2 -10755.436} C_VEL
LIN {X 0,Y 407.666,Z 429.083,A -85,B 0,C 180,E1 -10756.062,E2 -10756.062} C_VEL
LIN {X 0,Y 407.097,Z 440.615,A -85,B 0,C 180,E1 -10756.838,E2 -10756.838} C_VEL
LIN {X 0,Y 406.399,Z 452.575,A -85,B 0,C 180,E1 -10757.873,E2 -10757.873} C_VEL
LIN {X 0,Y 405.747,Z 462.662,A -85,B 0,C 180,E1 -10758.964,E2 -10758.964} C_VEL
LIN {X 0,Y 405.11,Z 472.114,A -85,B 0,C 180,E1 -10760.23,E2 -10760.23} C_VEL
LIN {X 0,Y 404.533,Z 480.775,A -85,B 0,C 180,E1 -10761.659,E2 -10761.659} C_VEL
LIN {X 0,Y 404.001,Z 488.051,A -85,B 0,C 180,E1 -10763.14,E2 -10763.14} C_VEL
LIN {X 0,Y 403.633,Z 493.877,A -85,B 0,C 180,E1 -10764.624,E2 -10764.624} C_VEL
LIN {X 0,Y 403.346,Z 498.482,A -85,B 0,C 180,E1 -10766.112,E2 -10766.112} C_VEL
LIN {X 0,Y 403.108,Z 502.511,A -85,B 0,C 180,E1 -10767.877,E2 -10767.877} C_VEL
LIN {X 0,Y 402.878,Z 505.143,A -85,B 0,C 180,E1 -10769.61,E2 -10769.61} C_VEL
LIN {X 0,Y 402.86,Z 506.202,A -85,B 0,C 180,E1 -10770.761,E2 -10770.761} C_VEL
LIN {X 0,Y 402.839,Z 506.675,A -85,B 0,C 180,E1 -10771.898,E2 -10771.898} C_VEL
LIN {X 0,Y 402.863,Z 506.667,A -85,B 0,C 180,E1 -10773.027,E2 -10773.027} C_VEL
LIN {X 0,Y 402.938,Z 506.092,A -85,B 0,C 180,E1 -10774.149,E2 -10774.149} C_VEL
LIN {X 0,Y 403.044,Z 505.041,A -85,B 0,C 180,E1 -10775.261,E2 -10775.261} C_VEL
LIN {X 0,Y 403.204,Z 503.47,A -85,B 0,C 180,E1 -10776.366,E2 -10776.366} C_VEL
LIN {X 0,Y 403.502,Z 500.142,A -85,B 0,C 180,E1 -10778.009,E2 -10778.009} C_VEL
LIN {X 0,Y 403.841,Z 495.605,A -85,B 0,C 180,E1 -10779.632,E2 -10779.632} C_VEL
LIN {X 0,Y 404.364,Z 489.715,A -85,B 0,C 180,E1 -10781.245,E2 -10781.245} C_VEL
LIN {X 0,Y 405.017,Z 482.24,A -85,B 0,C 180,E1 -10782.844,E2 -10782.844} C_VEL
LIN {X 0,Y 405.684,Z 474.551,A -85,B 0,C 180,E1 -10784.167,E2 -10784.167} C_VEL
LIN {X 0,Y 406.482,Z 465.113,A -85,B 0,C 180,E1 -10785.49,E2 -10785.49} C_VEL
LIN {X 0,Y 407.342,Z 454.749,A -85,B 0,C 180,E1 -10786.659,E2 -10786.659} C_VEL
LIN {X 0,Y 408.115,Z 443.163,A -85,B 0,C 180,E1 -10787.696,E2 -10787.696} C_VEL
LIN {X 0,Y 408.812,Z 431.399,A -85,B 0,C 180,E1 -10788.519,E2 -10788.519} C_VEL
LIN {X 0,Y 409.329,Z 418.823,A -85,B 0,C 180,E1 -10789.177,E2 -10789.177} C_VEL
LIN {X 0,Y 409.745,Z 405.454,A -85,B 0,C 180,E1 -10789.656,E2 -10789.656} C_VEL
LIN {X 0,Y 411.553,Z 315.097,A -85,B 0,C 180,E1 -10791.531,E2 -10791.531} C_VEL
LIN {X 0,Y 409.428,Z 305.399,A -85,B 0,C 180,E1 -10791.875,E2 -10791.875} C_VEL
LIN {X 0,Y 405.759,Z 296.082,A -85,B 0,C 180,E1 -10792.349,E2 -10792.349} C_VEL
LIN {X 0,Y 404.355,Z 290.12,A -85,B 0,C 180,E1 -10793.576,E2 -10793.576} C_VEL
LIN {X 0,Y 404.429,Z 290.11,A -85,B 0,C 180,E1 -10798.009,E2 -10798.009} C_VEL
LIN {X 0,Y 404.556,Z 290.091,A -85,B 0,C 180,E1 -10800,E2 -10800} C_VEL
LIN {X 0,Y 404.374,Z 290.116,A -85,B 0,C 180,E1 -10802.989,E2 -10802.989} C_VEL
LIN {X 0,Y 404.351,Z 290.12,A -85,B 0,C 180,E1 -10806.989,E2 -10806.989} C_VEL
LIN {X 0,Y 404.212,Z 290.132,A -85,B 0,C 180,E1 -10810.013,E2 -10810.013} C_VEL
LIN {X 0,Y 404.218,Z 290.134,A -85,B 0,C 180,E1 -10813.213,E2 -10813.213} C_VEL
LIN {X 0,Y 404.169,Z 290.139,A -85,B 0,C 180,E1 -10817.009,E2 -10817.009} C_VEL
LIN {X 0,Y 404.109,Z 290.142,A -85,B 0,C 180,E1 -10820.355,E2 -10820.355} C_VEL
LIN {X 0,Y 404.124,Z 290.145,A -85,B 0,C 180,E1 -10823.578,E2 -10823.578} C_VEL
LIN {X 0,Y 404.141,Z 290.138,A -85,B 0,C 180,E1 -10825.77,E2 -10825.77} C_VEL
LIN {X 0,Y 404.154,Z 290.139,A -85,B 0,C 180,E1 -10828.003,E2 -10828.003} C_VEL
LIN {X 0,Y 404.099,Z 290.145,A -85,B 0,C 180,E1 -10831.561,E2 -10831.561} C_VEL
LIN {X 0,Y 404.148,Z 290.14,A -85,B 0,C 180,E1 -10835.02,E2 -10835.02} C_VEL
LIN {X 0,Y 404.13,Z 290.145,A -85,B 0,C 180,E1 -10838.76,E2 -10838.76} C_VEL
LIN {X 0,Y 404.12,Z 290.144,A -85,B 0,C 180,E1 -10841.608,E2 -10841.608} C_VEL
LIN {X 0,Y 404.117,Z 290.144,A -85,B 0,C 180,E1 -10844.526,E2 -10844.526} C_VEL
LIN {X 0,Y 404.11,Z 290.149,A -85,B 0,C 180,E1 -10847.3,E2 -10847.3} C_VEL
LIN {X 0,Y 404.132,Z 290.143,A -85,B 0,C 180,E1 -10849.958,E2 -10849.958} C_VEL
LIN {X 0,Y 404.115,Z 290.15,A -85,B 0,C 180,E1 -10853.13,E2 -10853.13} C_VEL
LIN {X 0,Y 404.128,Z 290.15,A -85,B 0,C 180,E1 -10856.192,E2 -10856.192} C_VEL
LIN {X 0,Y 404.13,Z 290.153,A -85,B 0,C 180,E1 -10859.719,E2 -10859.719} C_VEL
LIN {X 0,Y 404.202,Z 290.227,A -85,B 0,C 180,E1 -10861.121,E2 -10861.121} C_VEL
LIN {X 0,Y 406.89,Z 302.169,A -85,B 0,C 180,E1 -10863.572,E2 -10863.572} C_VEL
LIN {X 0,Y 407.669,Z 306.734,A -85,B 0,C 180,E1 -10864.474,E2 -10864.474} C_VEL
LIN {X 0,Y 406.778,Z 321.403,A -85,B 0,C 180,E1 -10867.128,E2 -10867.128} C_VEL
LIN {X 0,Y 405.968,Z 336.037,A -85,B 0,C 180,E1 -10869.747,E2 -10869.747} C_VEL
LIN {X 0,Y 409.604,Z 358.133,A -85,B 0,C 180,E1 -10870.461,E2 -10870.461} C_VEL
LIN {X 0,Y 410.84,Z 369.392,A -85,B 0,C 180,E1 -10870.778,E2 -10870.778} C_VEL
LIN {X 0,Y 409.29,Z 447.711,A -85,B 0,C 180,E1 -10872.387,E2 -10872.387} C_VEL
LIN {X 0,Y 408.611,Z 461.508,A -85,B 0,C 180,E1 -10872.873,E2 -10872.873} C_VEL
LIN {X 0,Y 407.883,Z 473.433,A -85,B 0,C 180,E1 -10873.486,E2 -10873.486} C_VEL
LIN {X 0,Y 406.964,Z 485.97,A -85,B 0,C 180,E1 -10874.349,E2 -10874.349} C_VEL
LIN {X 0,Y 406.13,Z 497.252,A -85,B 0,C 180,E1 -10875.343,E2 -10875.343} C_VEL
LIN {X 0,Y 405.264,Z 508.211,A -85,B 0,C 180,E1 -10876.561,E2 -10876.561} C_VEL
LIN {X 0,Y 404.495,Z 518.391,A -85,B 0,C 180,E1 -10877.969,E2 -10877.969} C_VEL
LIN {X 0,Y 403.759,Z 527.107,A -85,B 0,C 180,E1 -10879.472,E2 -10879.472} C_VEL
LIN {X 0,Y 403.349,Z 534.129,A -85,B 0,C 180,E1 -10880.98,E2 -10880.98} C_VEL
LIN {X 0,Y 403.097,Z 539.776,A -85,B 0,C 180,E1 -10882.489,E2 -10882.489} C_VEL
LIN {X 0,Y 402.938,Z 544.202,A -85,B 0,C 180,E1 -10883.995,E2 -10883.995} C_VEL
LIN {X 0,Y 402.961,Z 546.562,A -85,B 0,C 180,E1 -10884.999,E2 -10884.999} C_VEL
LIN {X 0,Y 402.887,Z 548.414,A -85,B 0,C 180,E1 -10886.001,E2 -10886.001} C_VEL
LIN {X 0,Y 402.921,Z 549.836,A -85,B 0,C 180,E1 -10887.002,E2 -10887.002} C_VEL
LIN {X 0,Y 402.976,Z 550.852,A -85,B 0,C 180,E1 -10888.003,E2 -10888.003} C_VEL
LIN {X 0,Y 402.939,Z 551.442,A -85,B 0,C 180,E1 -10889.002,E2 -10889.002} C_VEL
LIN {X 0,Y 402.958,Z 551.58,A -85,B 0,C 180,E1 -10890.002,E2 -10890.002} C_VEL
LIN {X 0,Y 402.95,Z 551.31,A -85,B 0,C 180,E1 -10891.001,E2 -10891.001} C_VEL
LIN {X 0,Y 402.979,Z 550.639,A -85,B 0,C 180,E1 -10892,E2 -10892} C_VEL
LIN {X 0,Y 402.954,Z 549.529,A -85,B 0,C 180,E1 -10893.001,E2 -10893.001} C_VEL
LIN {X 0,Y 402.94,Z 547.032,A -85,B 0,C 180,E1 -10894.503,E2 -10894.503} C_VEL
LIN {X 0,Y 403.02,Z 542.681,A -85,B 0,C 180,E1 -10896.284,E2 -10896.284} C_VEL
LIN {X 0,Y 403.179,Z 536.928,A -85,B 0,C 180,E1 -10898.017,E2 -10898.017} C_VEL
LIN {X 0,Y 403.466,Z 530.493,A -85,B 0,C 180,E1 -10899.526,E2 -10899.526} C_VEL
LIN {X 0,Y 403.929,Z 522.403,A -85,B 0,C 180,E1 -10901.034,E2 -10901.034} C_VEL
LIN {X 0,Y 404.483,Z 514.153,A -85,B 0,C 180,E1 -10902.29,E2 -10902.29} C_VEL
LIN {X 0,Y 405.105,Z 505.427,A -85,B 0,C 180,E1 -10903.388,E2 -10903.388} C_VEL
LIN {X 0,Y 405.705,Z 495.498,A -85,B 0,C 180,E1 -10904.42,E2 -10904.42} C_VEL
LIN {X 0,Y 406.396,Z 485.137,A -85,B 0,C 180,E1 -10905.291,E2 -10905.291} C_VEL
LIN {X 0,Y 407.113,Z 472.815,A -85,B 0,C 180,E1 -10906.098,E2 -10906.098} C_VEL
LIN {X 0,Y 407.788,Z 459.269,A -85,B 0,C 180,E1 -10906.746,E2 -10906.746} C_VEL
LIN {X 0,Y 408.293,Z 446.719,A -85,B 0,C 180,E1 -10907.144,E2 -10907.144} C_VEL
LIN {X 0,Y 409.422,Z 367.449,A -85,B 0,C 180,E1 -10908.702,E2 -10908.702} C_VEL
LIN {X 0,Y 405.577,Z 339.125,A -85,B 0,C 180,E1 -10909.452,E2 -10909.452} C_VEL
LIN {X 0,Y 406.848,Z 319.777,A -85,B 0,C 180,E1 -10913.14,E2 -10913.14} C_VEL
LIN {X 0,Y 407.645,Z 307.382,A -85,B 0,C 180,E1 -10915.531,E2 -10915.531} C_VEL
LIN {X 0,Y 404.836,Z 293.254,A -85,B 0,C 180,E1 -10918.515,E2 -10918.515} C_VEL
LIN {X 0,Y 404.18,Z 290.138,A -85,B 0,C 180,E1 -10919.192,E2 -10919.192} C_VEL
LIN {X 0,Y 404.135,Z 290.147,A -85,B 0,C 180,E1 -10922.62,E2 -10922.62} C_VEL
LIN {X 0,Y 404.138,Z 290.142,A -85,B 0,C 180,E1 -10925.18,E2 -10925.18} C_VEL
LIN {X 0,Y 404.124,Z 290.148,A -85,B 0,C 180,E1 -10928.758,E2 -10928.758} C_VEL
LIN {X 0,Y 404.096,Z 290.146,A -85,B 0,C 180,E1 -10931.595,E2 -10931.595} C_VEL
LIN {X 0,Y 404.131,Z 290.145,A -85,B 0,C 180,E1 -10934.519,E2 -10934.519} C_VEL
LIN {X 0,Y 404.107,Z 290.146,A -85,B 0,C 180,E1 -10937.291,E2 -10937.291} C_VEL
LIN {X 0,Y 404.118,Z 290.143,A -85,B 0,C 180,E1 -10939.949,E2 -10939.949} C_VEL
LIN {X 0,Y 404.115,Z 290.147,A -85,B 0,C 180,E1 -10943.124,E2 -10943.124} C_VEL
LIN {X 0,Y 404.118,Z 290.144,A -85,B 0,C 180,E1 -10946.185,E2 -10946.185} C_VEL
LIN {X 0,Y 404.123,Z 290.144,A -85,B 0,C 180,E1 -10949.712,E2 -10949.712} C_VEL
LIN {X 0,Y 404.13,Z 290.146,A -85,B 0,C 180,E1 -10953.118,E2 -10953.118} C_VEL
LIN {X 0,Y 404.128,Z 290.143,A -85,B 0,C 180,E1 -10956.422,E2 -10956.422} C_VEL
LIN {X 0,Y 404.13,Z 290.144,A -85,B 0,C 180,E1 -10959.887,E2 -10959.887} C_VEL
LIN {X 0,Y 404.195,Z 290.139,A -85,B 0,C 180,E1 -10962.989,E2 -10962.989} C_VEL
LIN {X 0,Y 404.256,Z 290.13,A -85,B 0,C 180,E1 -10966.938,E2 -10966.938} C_VEL
LIN {X 0,Y 404.23,Z 290.132,A -85,B 0,C 180,E1 -10969.987,E2 -10969.987} C_VEL
LIN {X 0,Y 404.373,Z 290.116,A -85,B 0,C 180,E1 -10973.012,E2 -10973.012} C_VEL
LIN {X 0,Y 404.246,Z 290.132,A -85,B 0,C 180,E1 -10975.013,E2 -10975.013} C_VEL
LIN {X 0,Y 404.446,Z 290.105,A -85,B 0,C 180,E1 -10978.008,E2 -10978.008} C_VEL
LIN {X 0,Y 404.576,Z 290.089,A -85,B 0,C 180,E1 -10980,E2 -10980} C_VEL
LIN {X 0,Y 404.382,Z 290.114,A -85,B 0,C 180,E1 -10982.988,E2 -10982.988} C_VEL
LIN {X 0,Y 404.359,Z 290.115,A -85,B 0,C 180,E1 -10986.716,E2 -10986.716} C_VEL
LIN {X 0,Y 404.262,Z 290.128,A -85,B 0,C 180,E1 -10989.001,E2 -10989.001} C_VEL
LIN {X 0,Y 404.239,Z 290.131,A -85,B 0,C 180,E1 -10992.041,E2 -10992.041} C_VEL
LIN {X 0,Y 404.176,Z 290.139,A -85,B 0,C 180,E1 -10995.119,E2 -10995.119} C_VEL
LIN {X 0,Y 404.18,Z 290.139,A -85,B 0,C 180,E1 -10998.239,E2 -10998.239} C_VEL
LIN {X 0,Y 404.109,Z 290.149,A -85,B 0,C 180,E1 -11001.42,E2 -11001.42} C_VEL
LIN {X 0,Y 404.151,Z 290.141,A -85,B 0,C 180,E1 -11004.667,E2 -11004.667} C_VEL
LIN {X 0,Y 404.173,Z 290.14,A -85,B 0,C 180,E1 -11008.001,E2 -11008.001} C_VEL
LIN {X 0,Y 404.118,Z 290.147,A -85,B 0,C 180,E1 -11011.559,E2 -11011.559} C_VEL
LIN {X 0,Y 404.163,Z 290.14,A -85,B 0,C 180,E1 -11015.018,E2 -11015.018} C_VEL
LIN {X 0,Y 404.143,Z 290.142,A -85,B 0,C 180,E1 -11018.757,E2 -11018.757} C_VEL
LIN {X 0,Y 404.131,Z 290.146,A -85,B 0,C 180,E1 -11021.605,E2 -11021.605} C_VEL
LIN {X 0,Y 404.134,Z 290.145,A -85,B 0,C 180,E1 -11024.524,E2 -11024.524} C_VEL
LIN {X 0,Y 404.191,Z 290.136,A -85,B 0,C 180,E1 -11027.306,E2 -11027.306} C_VEL
LIN {X 0,Y 404.156,Z 290.142,A -85,B 0,C 180,E1 -11029.957,E2 -11029.957} C_VEL
LIN {X 0,Y 404.129,Z 290.144,A -85,B 0,C 180,E1 -11033.126,E2 -11033.126} C_VEL
LIN {X 0,Y 404.135,Z 290.144,A -85,B 0,C 180,E1 -11036.189,E2 -11036.189} C_VEL
LIN {X 0,Y 404.137,Z 290.144,A -85,B 0,C 180,E1 -11039.716,E2 -11039.716} C_VEL
LIN {X 0,Y 404.188,Z 290.136,A -85,B 0,C 180,E1 -11043.124,E2 -11043.124} C_VEL
LIN {X 0,Y 404.171,Z 290.138,A -85,B 0,C 180,E1 -11045.335,E2 -11045.335} C_VEL
LIN {X 0,Y 404.134,Z 290.146,A -85,B 0,C 180,E1 -11048.581,E2 -11048.581} C_VEL
LIN {X 0,Y 404.206,Z 290.135,A -85,B 0,C 180,E1 -11051.762,E2 -11051.762} C_VEL
LIN {X 0,Y 404.203,Z 290.137,A -85,B 0,C 180,E1 -11054.882,E2 -11054.882} C_VEL
LIN {X 0,Y 404.254,Z 290.129,A -85,B 0,C 180,E1 -11057.958,E2 -11057.958} C_VEL
LIN {X 0,Y 404.431,Z 290.106,A -85,B 0,C 180,E1 -11062.099,E2 -11062.099} C_VEL
LIN {X 0,Y 404.422,Z 290.108,A -85,B 0,C 180,E1 -11064.014,E2 -11064.014} C_VEL
LIN {X 0,Y 404.48,Z 290.1,A -85,B 0,C 180,E1 -11068.007,E2 -11068.007} C_VEL
LIN {X 0,Y 404.609,Z 290.084,A -85,B 0,C 180,E1 -11069.998,E2 -11069.998} C_VEL
LIN {X 0,Y 404.42,Z 290.11,A -85,B 0,C 180,E1 -11072.987,E2 -11072.987} C_VEL
LIN {X 0,Y 404.402,Z 290.113,A -85,B 0,C 180,E1 -11076.985,E2 -11076.985} C_VEL
LIN {X 0,Y 404.256,Z 290.127,A -85,B 0,C 180,E1 -11080.009,E2 -11080.009} C_VEL
LIN {X 0,Y 404.259,Z 290.129,A -85,B 0,C 180,E1 -11083.209,E2 -11083.209} C_VEL
LIN {X 0,Y 404.206,Z 290.138,A -85,B 0,C 180,E1 -11087.004,E2 -11087.004} C_VEL
LIN {X 0,Y 404.193,Z 290.135,A -85,B 0,C 180,E1 -11090.346,E2 -11090.346} C_VEL
LIN {X 0,Y 404.159,Z 290.138,A -85,B 0,C 180,E1 -11091.944,E2 -11091.944} C_VEL
LIN {X 0,Y 403.498,Z 290.225,A -85,B 0,C 180,E1 -11092.776,E2 -11092.776} C_VEL
LIN {X 0,Y 400.649,Z 290.578,A -85,B 0,C 180,E1 -11094.127,E2 -11094.127} C_VEL
LIN {X 0,Y 398.235,Z 290.88,A -85,B 0,C 180,E1 -11095.219,E2 -11095.219} C_VEL
LIN {X 0,Y 397.201,Z 291.006,A -85,B 0,C 180,E1 -11096.062,E2 -11096.062} C_VEL
LIN {X 0,Y 397.118,Z 291.015,A -85,B 0,C 180,E1 -11096.348,E2 -11096.348} C_VEL
LIN {X 0,Y 397.109,Z 291.017,A -85,B 0,C 180,E1 -11098.54,E2 -11098.54} C_VEL
LIN {X 0,Y 397.063,Z 291.021,A -85,B 0,C 180,E1 -11102.067,E2 -11102.067} C_VEL
LIN {X 0,Y 397.097,Z 291.02,A -85,B 0,C 180,E1 -11105.5,E2 -11105.5} C_VEL
LIN {X 0,Y 397.112,Z 291.018,A -85,B 0,C 180,E1 -11108.859,E2 -11108.859} C_VEL
LIN {X 0,Y 397.149,Z 291.093,A -85,B 0,C 180,E1 -11111.104,E2 -11111.104} C_VEL
LIN {X 0,Y 398.123,Z 295.928,A -85,B 0,C 180,E1 -11112.314,E2 -11112.314} C_VEL
LIN {X 0,Y 401.113,Z 306.1,A -85,B 0,C 180,E1 -11112.672,E2 -11112.672} C_VEL
LIN {X 0,Y 403.15,Z 316.346,A -85,B 0,C 180,E1 -11112.976,E2 -11112.976} C_VEL
LIN {X 0,Y 401.619,Z 403.865,A -85,B 0,C 180,E1 -11114.737,E2 -11114.737} C_VEL
LIN {X 0,Y 401.26,Z 417.413,A -85,B 0,C 180,E1 -11115.218,E2 -11115.218} C_VEL
LIN {X 0,Y 400.715,Z 430.266,A -85,B 0,C 180,E1 -11115.884,E2 -11115.884} C_VEL
LIN {X 0,Y 400.079,Z 442.662,A -85,B 0,C 180,E1 -11116.758,E2 -11116.758} C_VEL
LIN {X 0,Y 399.363,Z 454.436,A -85,B 0,C 180,E1 -11117.823,E2 -11117.823} C_VEL
LIN {X 0,Y 398.701,Z 464.402,A -85,B 0,C 180,E1 -11118.959,E2 -11118.959} C_VEL
LIN {X 0,Y 397.978,Z 474.382,A -85,B 0,C 180,E1 -11120.362,E2 -11120.362} C_VEL
LIN {X 0,Y 397.417,Z 482.435,A -85,B 0,C 180,E1 -11121.761,E2 -11121.761} C_VEL
LIN {X 0,Y 396.902,Z 489.56,A -85,B 0,C 180,E1 -11123.301,E2 -11123.301} C_VEL
LIN {X 0,Y 396.479,Z 495.826,A -85,B 0,C 180,E1 -11125.019,E2 -11125.019} C_VEL
LIN {X 0,Y 396.22,Z 500.357,A -85,B 0,C 180,E1 -11126.643,E2 -11126.643} C_VEL
LIN {X 0,Y 395.922,Z 503.926,A -85,B 0,C 180,E1 -11128.422,E2 -11128.422} C_VEL
LIN {X 0,Y 395.791,Z 506.35,A -85,B 0,C 180,E1 -11130.455,E2 -11130.455} C_VEL
LIN {X 0,Y 395.745,Z 506.904,A -85,B 0,C 180,E1 -11131.348,E2 -11131.348} C_VEL
LIN {X 0,Y 395.771,Z 507.131,A -85,B 0,C 180,E1 -11132.594,E2 -11132.594} C_VEL
LIN {X 0,Y 395.803,Z 506.851,A -85,B 0,C 180,E1 -11133.647,E2 -11133.647} C_VEL
LIN {X 0,Y 395.929,Z 506.009,A -85,B 0,C 180,E1 -11134.845,E2 -11134.845} C_VEL
LIN {X 0,Y 396.043,Z 504.748,A -85,B 0,C 180,E1 -11135.912,E2 -11135.912} C_VEL
LIN {X 0,Y 396.277,Z 502.562,A -85,B 0,C 180,E1 -11137.235,E2 -11137.235} C_VEL
LIN {X 0,Y 396.569,Z 499.252,A -85,B 0,C 180,E1 -11138.698,E2 -11138.698} C_VEL
LIN {X 0,Y 397.02,Z 494.261,A -85,B 0,C 180,E1 -11140.347,E2 -11140.347} C_VEL
LIN {X 0,Y 397.598,Z 487.871,A -85,B 0,C 180,E1 -11141.982,E2 -11141.982} C_VEL
LIN {X 0,Y 398.356,Z 479.835,A -85,B 0,C 180,E1 -11143.604,E2 -11143.604} C_VEL
LIN {X 0,Y 399.221,Z 470.351,A -85,B 0,C 180,E1 -11145.112,E2 -11145.112} C_VEL
LIN {X 0,Y 400.149,Z 460.164,A -85,B 0,C 180,E1 -11146.414,E2 -11146.414} C_VEL
LIN {X 0,Y 400.944,Z 449.837,A -85,B 0,C 180,E1 -11147.473,E2 -11147.473} C_VEL
LIN {X 0,Y 401.711,Z 438.412,A -85,B 0,C 180,E1 -11148.407,E2 -11148.407} C_VEL
LIN {X 0,Y 402.411,Z 426.166,A -85,B 0,C 180,E1 -11149.179,E2 -11149.179} C_VEL
LIN {X 0,Y 402.888,Z 413.282,A -85,B 0,C 180,E1 -11149.764,E2 -11149.764} C_VEL
LIN {X 0,Y 403.281,Z 399.919,A -85,B 0,C 180,E1 -11150.154,E2 -11150.154} C_VEL
LIN {X 0,Y 405.07,Z 316.305,A -85,B 0,C 180,E1 -11151.903,E2 -11151.903} C_VEL
LIN {X 0,Y 403.079,Z 307.458,A -85,B 0,C 180,E1 -11152.235,E2 -11152.235} C_VEL
LIN {X 0,Y 398.714,Z 296.714,A -85,B 0,C 180,E1 -11152.786,E2 -11152.786} C_VEL
LIN {X 0,Y 397.327,Z 290.997,A -85,B 0,C 180,E1 -11153.972,E2 -11153.972} C_VEL
LIN {X 0,Y 397.398,Z 290.986,A -85,B 0,C 180,E1 -11157.974,E2 -11157.974} C_VEL
LIN {X 0,Y 397.526,Z 290.967,A -85,B 0,C 180,E1 -11160,E2 -11160} C_VEL
LIN {X 0,Y 397.333,Z 290.993,A -85,B 0,C 180,E1 -11163.042,E2 -11163.042} C_VEL
LIN {X 0,Y 397.302,Z 290.999,A -85,B 0,C 180,E1 -11167.113,E2 -11167.113} C_VEL
LIN {X 0,Y 397.173,Z 291.009,A -85,B 0,C 180,E1 -11170.193,E2 -11170.193} C_VEL
LIN {X 0,Y 397.179,Z 291.012,A -85,B 0,C 180,E1 -11173.323,E2 -11173.323} C_VEL
LIN {X 0,Y 397.135,Z 291.014,A -85,B 0,C 180,E1 -11177.157,E2 -11177.157} C_VEL
LIN {X 0,Y 397.052,Z 291.022,A -85,B 0,C 180,E1 -11180.733,E2 -11180.733} C_VEL
LIN {X 0,Y 397.088,Z 291.019,A -85,B 0,C 180,E1 -11184.022,E2 -11184.022} C_VEL
LIN {X 0,Y 397.153,Z 291.015,A -85,B 0,C 180,E1 -11187.394,E2 -11187.394} C_VEL
LIN {X 0,Y 397.039,Z 291.029,A -85,B 0,C 180,E1 -11190.886,E2 -11190.886} C_VEL
LIN {X 0,Y 397.089,Z 291.017,A -85,B 0,C 180,E1 -11194.497,E2 -11194.497} C_VEL
LIN {X 0,Y 397.076,Z 291.021,A -85,B 0,C 180,E1 -11198.279,E2 -11198.279} C_VEL
LIN {X 0,Y 397.082,Z 291.023,A -85,B 0,C 180,E1 -11200.91,E2 -11200.91} C_VEL
LIN {X 0,Y 397.074,Z 291.023,A -85,B 0,C 180,E1 -11203.653,E2 -11203.653} C_VEL
LIN {X 0,Y 397.076,Z 291.022,A -85,B 0,C 180,E1 -11206.526,E2 -11206.526} C_VEL
LIN {X 0,Y 397.081,Z 291.021,A -85,B 0,C 180,E1 -11210.426,E2 -11210.426} C_VEL
LIN {X 0,Y 397.089,Z 291.024,A -85,B 0,C 180,E1 -11214.27,E2 -11214.27} C_VEL
LIN {X 0,Y 397.098,Z 291.027,A -85,B 0,C 180,E1 -11216.731,E2 -11216.731} C_VEL
LIN {X 0,Y 397.141,Z 291.112,A -85,B 0,C 180,E1 -11220.739,E2 -11220.739} C_VEL
LIN {X 0,Y 399.915,Z 303.217,A -85,B 0,C 180,E1 -11223.291,E2 -11223.291} C_VEL
LIN {X 0,Y 400.811,Z 308.11,A -85,B 0,C 180,E1 -11224.284,E2 -11224.284} C_VEL
LIN {X 0,Y 399.9,Z 322.779,A -85,B 0,C 180,E1 -11226.986,E2 -11226.986} C_VEL
LIN {X 0,Y 399.138,Z 335.541,A -85,B 0,C 180,E1 -11229.306,E2 -11229.306} C_VEL
LIN {X 0,Y 402.64,Z 356.068,A -85,B 0,C 180,E1 -11230.001,E2 -11230.001} C_VEL
LIN {X 0,Y 404.284,Z 369.591,A -85,B 0,C 180,E1 -11230.401,E2 -11230.401} C_VEL
LIN {X 0,Y 402.671,Z 446.699,A -85,B 0,C 180,E1 -11232.022,E2 -11232.022} C_VEL
LIN {X 0,Y 401.928,Z 460.591,A -85,B 0,C 180,E1 -11232.514,E2 -11232.514} C_VEL
LIN {X 0,Y 401.09,Z 473.603,A -85,B 0,C 180,E1 -11233.198,E2 -11233.198} C_VEL
LIN {X 0,Y 400.118,Z 485.984,A -85,B 0,C 180,E1 -11234.074,E2 -11234.074} C_VEL
LIN {X 0,Y 399.239,Z 497.183,A -85,B 0,C 180,E1 -11235.084,E2 -11235.084} C_VEL
LIN {X 0,Y 398.403,Z 507.403,A -85,B 0,C 180,E1 -11236.238,E2 -11236.238} C_VEL
LIN {X 0,Y 397.683,Z 516.538,A -85,B 0,C 180,E1 -11237.5,E2 -11237.5} C_VEL
LIN {X 0,Y 396.866,Z 525.582,A -85,B 0,C 180,E1 -11239.028,E2 -11239.028} C_VEL
LIN {X 0,Y 396.369,Z 532.824,A -85,B 0,C 180,E1 -11240.563,E2 -11240.563} C_VEL
LIN {X 0,Y 396.031,Z 539.482,A -85,B 0,C 180,E1 -11242.354,E2 -11242.354} C_VEL
LIN {X 0,Y 395.834,Z 544.625,A -85,B 0,C 180,E1 -11244.186,E2 -11244.186} C_VEL
LIN {X 0,Y 395.808,Z 548.055,A -85,B 0,C 180,E1 -11245.929,E2 -11245.929} C_VEL
LIN {X 0,Y 395.821,Z 549.47,A -85,B 0,C 180,E1 -11246.949,E2 -11246.949} C_VEL
LIN {X 0,Y 395.904,Z 550.477,A -85,B 0,C 180,E1 -11247.967,E2 -11247.967} C_VEL
LIN {X 0,Y 395.865,Z 551.046,A -85,B 0,C 180,E1 -11248.984,E2 -11248.984} C_VEL
LIN {X 0,Y 395.88,Z 551.172,A -85,B 0,C 180,E1 -11250.002,E2 -11250.002} C_VEL
LIN {X 0,Y 395.875,Z 550.891,A -85,B 0,C 180,E1 -11251.019,E2 -11251.019} C_VEL
LIN {X 0,Y 395.909,Z 550.207,A -85,B 0,C 180,E1 -11252.036,E2 -11252.036} C_VEL
LIN {X 0,Y 395.856,Z 549.066,A -85,B 0,C 180,E1 -11253.054,E2 -11253.054} C_VEL
LIN {X 0,Y 395.872,Z 546.541,A -85,B 0,C 180,E1 -11254.583,E2 -11254.583} C_VEL
LIN {X 0,Y 395.976,Z 541.643,A -85,B 0,C 180,E1 -11256.574,E2 -11256.574} C_VEL
LIN {X 0,Y 396.113,Z 536.354,A -85,B 0,C 180,E1 -11258.161,E2 -11258.161} C_VEL
LIN {X 0,Y 396.407,Z 529.854,A -85,B 0,C 180,E1 -11259.697,E2 -11259.697} C_VEL
LIN {X 0,Y 396.936,Z 521.704,A -85,B 0,C 180,E1 -11261.231,E2 -11261.231} C_VEL
LIN {X 0,Y 397.465,Z 513.381,A -85,B 0,C 180,E1 -11262.51,E2 -11262.51} C_VEL
LIN {X 0,Y 398.216,Z 503.648,A -85,B 0,C 180,E1 -11263.736,E2 -11263.736} C_VEL
LIN {X 0,Y 398.856,Z 493.173,A -85,B 0,C 180,E1 -11264.803,E2 -11264.803} C_VEL
LIN {X 0,Y 399.711,Z 480.516,A -85,B 0,C 180,E1 -11265.815,E2 -11265.815} C_VEL
LIN {X 0,Y 400.429,Z 468.024,A -85,B 0,C 180,E1 -11266.571,E2 -11266.571} C_VEL
LIN {X 0,Y 401.103,Z 454.921,A -85,B 0,C 180,E1 -11267.132,E2 -11267.132} C_VEL
LIN {X 0,Y 401.569,Z 441.146,A -85,B 0,C 180,E1 -11267.506,E2 -11267.506} C_VEL
LIN {X 0,Y 402.553,Z 367.871,A -85,B 0,C 180,E1 -11268.97,E2 -11268.97} C_VEL
LIN {X 0,Y 398.623,Z 338.781,A -85,B 0,C 180,E1 -11269.756,E2 -11269.756} C_VEL
LIN {X 0,Y 399.987,Z 319.168,A -85,B 0,C 180,E1 -11273.561,E2 -11273.561} C_VEL
LIN {X 0,Y 400.697,Z 309.549,A -85,B 0,C 180,E1 -11275.449,E2 -11275.449} C_VEL
LIN {X 0,Y 398.773,Z 298.711,A -85,B 0,C 180,E1 -11277.748,E2 -11277.748} C_VEL
LIN {X 0,Y 397.122,Z 291.017,A -85,B 0,C 180,E1 -11279.484,E2 -11279.484} C_VEL
LIN {X 0,Y 397.107,Z 291.017,A -85,B 0,C 180,E1 -11283.272,E2 -11283.272} C_VEL
LIN {X 0,Y 397.087,Z 291.022,A -85,B 0,C 180,E1 -11286.994,E2 -11286.994} C_VEL
LIN {X 0,Y 397.046,Z 291.027,A -85,B 0,C 180,E1 -11290.435,E2 -11290.435} C_VEL
LIN {X 0,Y 397.076,Z 291.021,A -85,B 0,C 180,E1 -11293.649,E2 -11293.649} C_VEL
LIN {X 0,Y 397.078,Z 291.023,A -85,B 0,C 180,E1 -11296.521,E2 -11296.521} C_VEL
LIN {X 0,Y 397.071,Z 291.023,A -85,B 0,C 180,E1 -11300.417,E2 -11300.417} C_VEL
LIN {X 0,Y 397.077,Z 291.025,A -85,B 0,C 180,E1 -11303.002,E2 -11303.002} C_VEL
LIN {X 0,Y 397.092,Z 291.023,A -85,B 0,C 180,E1 -11306.724,E2 -11306.724} C_VEL
LIN {X 0,Y 397.098,Z 291.019,A -85,B 0,C 180,E1 -11310.293,E2 -11310.293} C_VEL
LIN {X 0,Y 397.079,Z 291.022,A -85,B 0,C 180,E1 -11313.737,E2 -11313.737} C_VEL
LIN {X 0,Y 397.076,Z 291.025,A -85,B 0,C 180,E1 -11317.083,E2 -11317.083} C_VEL
LIN {X 0,Y 397.105,Z 291.018,A -85,B 0,C 180,E1 -11320.35,E2 -11320.35} C_VEL
LIN {X 0,Y 397.142,Z 291.015,A -85,B 0,C 180,E1 -11323.552,E2 -11323.552} C_VEL
LIN {X 0,Y 397.203,Z 291.007,A -85,B 0,C 180,E1 -11326.701,E2 -11326.701} C_VEL
LIN {X 0,Y 397.19,Z 291.009,A -85,B 0,C 180,E1 -11329.808,E2 -11329.808} C_VEL
LIN {X 0,Y 397.323,Z 290.993,A -85,B 0,C 180,E1 -11332.887,E2 -11332.887} C_VEL
LIN {X 0,Y 397.218,Z 291.006,A -85,B 0,C 180,E1 -11334.924,E2 -11334.924} C_VEL
LIN {X 0,Y 397.416,Z 290.981,A -85,B 0,C 180,E1 -11337.973,E2 -11337.973} C_VEL
LIN {X 0,Y 397.546,Z 290.965,A -85,B 0,C 180,E1 -11340,E2 -11340} C_VEL
LIN {X 0,Y 397.341,Z 290.991,A -85,B 0,C 180,E1 -11343.041,E2 -11343.041} C_VEL
LIN {X 0,Y 397.309,Z 290.993,A -85,B 0,C 180,E1 -11346.715,E2 -11346.715} C_VEL
LIN {X 0,Y 397.224,Z 291.006,A -85,B 0,C 180,E1 -11349.162,E2 -11349.162} C_VEL
LIN {X 0,Y 397.199,Z 291.008,A -85,B 0,C 180,E1 -11352.258,E2 -11352.258} C_VEL
LIN {X 0,Y 397.149,Z 291.016,A -85,B 0,C 180,E1 -11355.393,E2 -11355.393} C_VEL
LIN {X 0,Y 397.132,Z 291.015,A -85,B 0,C 180,E1 -11358.574,E2 -11358.574} C_VEL
LIN {X 0,Y 397.068,Z 291.025,A -85,B 0,C 180,E1 -11361.82,E2 -11361.82} C_VEL
LIN {X 0,Y 397.131,Z 291.016,A -85,B 0,C 180,E1 -11365.133,E2 -11365.133} C_VEL
LIN {X 0,Y 397.139,Z 291.016,A -85,B 0,C 180,E1 -11367.777,E2 -11367.777} C_VEL
LIN {X 0,Y 397.059,Z 291.024,A -85,B 0,C 180,E1 -11370.884,E2 -11370.884} C_VEL
LIN {X 0,Y 397.104,Z 291.02,A -85,B 0,C 180,E1 -11374.495,E2 -11374.495} C_VEL
LIN {X 0,Y 397.09,Z 291.023,A -85,B 0,C 180,E1 -11378.276,E2 -11378.276} C_VEL
LIN {X 0,Y 397.094,Z 291.02,A -85,B 0,C 180,E1 -11380.907,E2 -11380.907} C_VEL
LIN {X 0,Y 397.086,Z 291.023,A -85,B 0,C 180,E1 -11383.65,E2 -11383.65} C_VEL
LIN {X 0,Y 397.142,Z 291.016,A -85,B 0,C 180,E1 -11386.514,E2 -11386.514} C_VEL
LIN {X 0,Y 397.11,Z 291.019,A -85,B 0,C 180,E1 -11389.552,E2 -11389.552} C_VEL
LIN {X 0,Y 397.087,Z 291.022,A -85,B 0,C 180,E1 -11392.791,E2 -11392.791} C_VEL
LIN {X 0,Y 397.109,Z 291.02,A -85,B 0,C 180,E1 -11396.283,E2 -11396.283} C_VEL
LIN {X 0,Y 397.097,Z 291.021,A -85,B 0,C 180,E1 -11400.136,E2 -11400.136} C_VEL
LIN {X 0,Y 397.187,Z 291.012,A -85,B 0,C 180,E1 -11402.611,E2 -11402.611} C_VEL
LIN {X 0,Y 397.127,Z 291.017,A -85,B 0,C 180,E1 -11405.982,E2 -11405.982} C_VEL
LIN {X 0,Y 397.134,Z 291.015,A -85,B 0,C 180,E1 -11409.705,E2 -11409.705} C_VEL
LIN {X 0,Y 397.179,Z 291.011,A -85,B 0,C 180,E1 -11412.845,E2 -11412.845} C_VEL
LIN {X 0,Y 397.226,Z 291.007,A -85,B 0,C 180,E1 -11416.702,E2 -11416.702} C_VEL
LIN {X 0,Y 397.216,Z 291.005,A -85,B 0,C 180,E1 -11419.808,E2 -11419.808} C_VEL
LIN {X 0,Y 397.362,Z 290.989,A -85,B 0,C 180,E1 -11422.887,E2 -11422.887} C_VEL
LIN {X 0,Y 397.252,Z 291.003,A -85,B 0,C 180,E1 -11424.924,E2 -11424.924} C_VEL
LIN {X 0,Y 397.449,Z 290.976,A -85,B 0,C 180,E1 -11427.972,E2 -11427.972} C_VEL
LIN {X 0,Y 397.578,Z 290.96,A -85,B 0,C 180,E1 -11429.998,E2 -11429.998} C_VEL
LIN {X 0,Y 397.378,Z 290.987,A -85,B 0,C 180,E1 -11433.039,E2 -11433.039} C_VEL
LIN {X 0,Y 397.355,Z 290.989,A -85,B 0,C 180,E1 -11437.11,E2 -11437.11} C_VEL
LIN {X 0,Y 397.216,Z 291.004,A -85,B 0,C 180,E1 -11440.188,E2 -11440.188} C_VEL
LIN {X 0,Y 397.219,Z 291.005,A -85,B 0,C 180,E1 -11443.318,E2 -11443.318} C_VEL
LIN {X 0,Y 397.172,Z 291.013,A -85,B 0,C 180,E1 -11447.152,E2 -11447.152} C_VEL
LIN {X 0,Y 397.142,Z 291.015,A -85,B 0,C 180,E1 -11450.724,E2 -11450.724} C_VEL
LIN {X 0,Y 397.12,Z 291.015,A -85,B 0,C 180,E1 -11454.015,E2 -11454.015} C_VEL
LIN {X 0,Y 397.118,Z 291.015,A -85,B 0,C 180,E1 -11456.348,E2 -11456.348} C_VEL
LIN {X 0,Y 396.45,Z 291.103,A -85,B 0,C 180,E1 -11457.195,E2 -11457.195} C_VEL
LIN {X 0,Y 393.575,Z 291.458,A -85,B 0,C 180,E1 -11458.57,E2 -11458.57} C_VEL
LIN {X 0,Y 391.137,Z 291.761,A -85,B 0,C 180,E1 -11459.682,E2 -11459.682} C_VEL
LIN {X 0,Y 390.086,Z 291.892,A -85,B 0,C 180,E1 -11460.542,E2 -11460.542} C_VEL
LIN {X 0,Y 389.998,Z 291.9,A -85,B 0,C 180,E1 -11460.833,E2 -11460.833} C_VEL
LIN {X 0,Y 390.046,Z 291.895,A -85,B 0,C 180,E1 -11464.021,E2 -11464.021} C_VEL
LIN {X 0,Y 390.022,Z 291.904,A -85,B 0,C 180,E1 -11467.548,E2 -11467.548} C_VEL
LIN {X 0,Y 390.108,Z 291.984,A -85,B 0,C 180,E1 -11470.903,E2 -11470.903} C_VEL
LIN {X 0,Y 391.006,Z 296.556,A -85,B 0,C 180,E1 -11472.014,E2 -11472.014} C_VEL
LIN {X 0,Y 394.522,Z 308.027,A -85,B 0,C 180,E1 -11472.423,E2 -11472.423} C_VEL
LIN {X 0,Y 396.33,Z 317.731,A -85,B 0,C 180,E1 -11472.712,E2 -11472.712} C_VEL
LIN {X 0,Y 394.711,Z 404.841,A -85,B 0,C 180,E1 -11474.512,E2 -11474.512} C_VEL
LIN {X 0,Y 394.38,Z 417.995,A -85,B 0,C 180,E1 -11474.995,E2 -11474.995} C_VEL
LIN {X 0,Y 393.781,Z 431.144,A -85,B 0,C 180,E1 -11475.696,E2 -11475.696} C_VEL
LIN {X 0,Y 393.176,Z 442.571,A -85,B 0,C 180,E1 -11476.514,E2 -11476.514} C_VEL
LIN {X 0,Y 392.493,Z 453.426,A -85,B 0,C 180,E1 -11477.496,E2 -11477.496} C_VEL
LIN {X 0,Y 391.761,Z 464.15,A -85,B 0,C 180,E1 -11478.708,E2 -11478.708} C_VEL
LIN {X 0,Y 391.087,Z 473.13,A -85,B 0,C 180,E1 -11479.962,E2 -11479.962} C_VEL
LIN {X 0,Y 390.503,Z 480.954,A -85,B 0,C 180,E1 -11481.289,E2 -11481.289} C_VEL
LIN {X 0,Y 389.914,Z 488.971,A -85,B 0,C 180,E1 -11482.965,E2 -11482.965} C_VEL
LIN {X 0,Y 389.461,Z 495.497,A -85,B 0,C 180,E1 -11484.729,E2 -11484.729} C_VEL
LIN {X 0,Y 389.213,Z 499.625,A -85,B 0,C 180,E1 -11486.151,E2 -11486.151} C_VEL
LIN {X 0,Y 389.074,Z 502.034,A -85,B 0,C 180,E1 -11487.187,E2 -11487.187} C_VEL
LIN {X 0,Y 388.835,Z 504.287,A -85,B 0,C 180,E1 -11488.389,E2 -11488.389} C_VEL
LIN {X 0,Y 388.701,Z 506.517,A -85,B 0,C 180,E1 -11490.199,E2 -11490.199} C_VEL
LIN {X 0,Y 388.682,Z 507.561,A -85,B 0,C 180,E1 -11492.36,E2 -11492.36} C_VEL
LIN {X 0,Y 388.792,Z 506.939,A -85,B 0,C 180,E1 -11494.289,E2 -11494.289} C_VEL
LIN {X 0,Y 388.9,Z 505.906,A -85,B 0,C 180,E1 -11495.441,E2 -11495.441} C_VEL
LIN {X 0,Y 389.206,Z 503.583,A -85,B 0,C 180,E1 -11497.043,E2 -11497.043} C_VEL
LIN {X 0,Y 389.543,Z 499.71,A -85,B 0,C 180,E1 -11498.849,E2 -11498.849} C_VEL
LIN {X 0,Y 390.03,Z 494.724,A -85,B 0,C 180,E1 -11500.528,E2 -11500.528} C_VEL
LIN {X 0,Y 390.64,Z 488.351,A -85,B 0,C 180,E1 -11502.191,E2 -11502.191} C_VEL
LIN {X 0,Y 391.453,Z 480.349,A -85,B 0,C 180,E1 -11503.843,E2 -11503.843} C_VEL
LIN {X 0,Y 392.32,Z 471.498,A -85,B 0,C 180,E1 -11505.291,E2 -11505.291} C_VEL
LIN {X 0,Y 393.225,Z 461.891,A -85,B 0,C 180,E1 -11506.565,E2 -11506.565} C_VEL
LIN {X 0,Y 394.122,Z 451.859,A -85,B 0,C 180,E1 -11507.645,E2 -11507.645} C_VEL
LIN {X 0,Y 394.919,Z 440.601,A -85,B 0,C 180,E1 -11508.612,E2 -11508.612} C_VEL
LIN {X 0,Y 395.655,Z 428.049,A -85,B 0,C 180,E1 -11509.445,E2 -11509.445} C_VEL
LIN {X 0,Y 396.207,Z 415.037,A -85,B 0,C 180,E1 -11510.074,E2 -11510.074} C_VEL
LIN {X 0,Y 396.655,Z 401.048,A -85,B 0,C 180,E1 -11510.503,E2 -11510.503} C_VEL
LIN {X 0,Y 398.637,Z 318.262,A -85,B 0,C 180,E1 -11512.278,E2 -11512.278} C_VEL
LIN {X 0,Y 397.081,Z 310.456,A -85,B 0,C 180,E1 -11512.57,E2 -11512.57} C_VEL
LIN {X 0,Y 391.636,Z 297.088,A -85,B 0,C 180,E1 -11513.302,E2 -11513.302} C_VEL
LIN {X 0,Y 390.228,Z 291.882,A -85,B 0,C 180,E1 -11514.445,E2 -11514.445} C_VEL
LIN {X 0,Y 390.368,Z 291.863,A -85,B 0,C 180,E1 -11517.937,E2 -11517.937} C_VEL
LIN {X 0,Y 390.496,Z 291.842,A -85,B 0,C 180,E1 -11520.001,E2 -11520.001} C_VEL
LIN {X 0,Y 390.267,Z 291.873,A -85,B 0,C 180,E1 -11523.097,E2 -11523.097} C_VEL
LIN {X 0,Y 390.274,Z 291.87,A -85,B 0,C 180,E1 -11526.203,E2 -11526.203} C_VEL
LIN {X 0,Y 390.157,Z 291.887,A -85,B 0,C 180,E1 -11529.33,E2 -11529.33} C_VEL
LIN {X 0,Y 390.13,Z 291.888,A -85,B 0,C 180,E1 -11532.485,E2 -11532.485} C_VEL
LIN {X 0,Y 390.091,Z 291.892,A -85,B 0,C 180,E1 -11535.679,E2 -11535.679} C_VEL
LIN {X 0,Y 390.053,Z 291.898,A -85,B 0,C 180,E1 -11538.925,E2 -11538.925} C_VEL
LIN {X 0,Y 389.993,Z 291.903,A -85,B 0,C 180,E1 -11542.237,E2 -11542.237} C_VEL
LIN {X 0,Y 390.077,Z 291.89,A -85,B 0,C 180,E1 -11545.746,E2 -11545.746} C_VEL
LIN {X 0,Y 390.017,Z 291.9,A -85,B 0,C 180,E1 -11549.113,E2 -11549.113} C_VEL
LIN {X 0,Y 390.005,Z 291.902,A -85,B 0,C 180,E1 -11552.726,E2 -11552.726} C_VEL
LIN {X 0,Y 390.022,Z 291.901,A -85,B 0,C 180,E1 -11555.829,E2 -11555.829} C_VEL
LIN {X 0,Y 390.043,Z 291.899,A -85,B 0,C 180,E1 -11559.223,E2 -11559.223} C_VEL
LIN {X 0,Y 390.026,Z 291.896,A -85,B 0,C 180,E1 -11562.38,E2 -11562.38} C_VEL
LIN {X 0,Y 390.017,Z 291.905,A -85,B 0,C 180,E1 -11565.358,E2 -11565.358} C_VEL
LIN {X 0,Y 390.006,Z 291.903,A -85,B 0,C 180,E1 -11568.191,E2 -11568.191} C_VEL
LIN {X 0,Y 390.061,Z 291.897,A -85,B 0,C 180,E1 -11570.911,E2 -11570.911} C_VEL
LIN {X 0,Y 390.067,Z 291.901,A -85,B 0,C 180,E1 -11574.797,E2 -11574.797} C_VEL
LIN {X 0,Y 390.008,Z 291.912,A -85,B 0,C 180,E1 -11578.5,E2 -11578.5} C_VEL
LIN {X 0,Y 390.06,Z 291.904,A -85,B 0,C 180,E1 -11580.303,E2 -11580.303} C_VEL
LIN {X 0,Y 392.852,Z 303.71,A -85,B 0,C 180,E1 -11582.864,E2 -11582.864} C_VEL
LIN {X 0,Y 393.968,Z 309.593,A -85,B 0,C 180,E1 -11584.088,E2 -11584.088} C_VEL
LIN {X 0,Y 393.102,Z 322.771,A -85,B 0,C 180,E1 -11586.564,E2 -11586.564} C_VEL
LIN {X 0,Y 392.315,Z 335.032,A -85,B 0,C 180,E1 -11588.835,E2 -11588.835} C_VEL
LIN {X 0,Y 396,Z 355.947,A -85,B 0,C 180,E1 -11589.58,E2 -11589.58} C_VEL
LIN {X 0,Y 397.696,Z 371.295,A -85,B 0,C 180,E1 -11590.048,E2 -11590.048} C_VEL
LIN {X 0,Y 396.036,Z 445.879,A -85,B 0,C 180,E1 -11591.643,E2 -11591.643} C_VEL
LIN {X 0,Y 395.29,Z 459.858,A -85,B 0,C 180,E1 -11592.143,E2 -11592.143} C_VEL
LIN {X 0,Y 394.468,Z 471.963,A -85,B 0,C 180,E1 -11592.774,E2 -11592.774} C_VEL
LIN {X 0,Y 393.434,Z 484.58,A -85,B 0,C 180,E1 -11593.663,E2 -11593.663} C_VEL
LIN {X 0,Y 392.464,Z 495.921,A -85,B 0,C 180,E1 -11594.688,E2 -11594.688} C_VEL
LIN {X 0,Y 391.562,Z 506.258,A -85,B 0,C 180,E1 -11595.854,E2 -11595.854} C_VEL
LIN {X 0,Y 390.722,Z 516.361,A -85,B 0,C 180,E1 -11597.274,E2 -11597.274} C_VEL
LIN {X 0,Y 389.849,Z 525.364,A -85,B 0,C 180,E1 -11598.828,E2 -11598.828} C_VEL
LIN {X 0,Y 389.322,Z 532.566,A -85,B 0,C 180,E1 -11600.39,E2 -11600.39} C_VEL
LIN {X 0,Y 388.964,Z 539.205,A -85,B 0,C 180,E1 -11602.214,E2 -11602.214} C_VEL
LIN {X 0,Y 388.776,Z 543.779,A -85,B 0,C 180,E1 -11603.856,E2 -11603.856} C_VEL
LIN {X 0,Y 388.763,Z 545.894,A -85,B 0,C 180,E1 -11604.816,E2 -11604.816} C_VEL
LIN {X 0,Y 388.731,Z 547.712,A -85,B 0,C 180,E1 -11605.855,E2 -11605.855} C_VEL
LIN {X 0,Y 388.816,Z 550.108,A -85,B 0,C 180,E1 -11607.93,E2 -11607.93} C_VEL
LIN {X 0,Y 388.793,Z 550.649,A -85,B 0,C 180,E1 -11608.966,E2 -11608.966} C_VEL
LIN {X 0,Y 388.804,Z 550.762,A -85,B 0,C 180,E1 -11610.002,E2 -11610.002} C_VEL
LIN {X 0,Y 388.803,Z 550.469,A -85,B 0,C 180,E1 -11611.037,E2 -11611.037} C_VEL
LIN {X 0,Y 388.84,Z 549.771,A -85,B 0,C 180,E1 -11612.073,E2 -11612.073} C_VEL
LIN {X 0,Y 388.759,Z 548.599,A -85,B 0,C 180,E1 -11613.11,E2 -11613.11} C_VEL
LIN {X 0,Y 388.803,Z 546.043,A -85,B 0,C 180,E1 -11614.667,E2 -11614.667} C_VEL
LIN {X 0,Y 388.837,Z 542.417,A -85,B 0,C 180,E1 -11616.227,E2 -11616.227} C_VEL
LIN {X 0,Y 388.97,Z 537.628,A -85,B 0,C 180,E1 -11617.789,E2 -11617.789} C_VEL
LIN {X 0,Y 389.235,Z 531.536,A -85,B 0,C 180,E1 -11619.353,E2 -11619.353} C_VEL
LIN {X 0,Y 389.655,Z 523.923,A -85,B 0,C 180,E1 -11620.917,E2 -11620.917} C_VEL
LIN {X 0,Y 390.282,Z 516.161,A -85,B 0,C 180,E1 -11622.216,E2 -11622.216} C_VEL
LIN {X 0,Y 390.974,Z 506.703,A -85,B 0,C 180,E1 -11623.514,E2 -11623.514} C_VEL
LIN {X 0,Y 391.662,Z 496.17,A -85,B 0,C 180,E1 -11624.683,E2 -11624.683} C_VEL
LIN {X 0,Y 392.463,Z 484.521,A -85,B 0,C 180,E1 -11625.715,E2 -11625.715} C_VEL
LIN {X 0,Y 393.234,Z 472.261,A -85,B 0,C 180,E1 -11626.549,E2 -11626.549} C_VEL
LIN {X 0,Y 393.989,Z 458.82,A -85,B 0,C 180,E1 -11627.217,E2 -11627.217} C_VEL
LIN {X 0,Y 394.524,Z 446.571,A -85,B 0,C 180,E1 -11627.628,E2 -11627.628} C_VEL
LIN {X 0,Y 395.803,Z 369.297,A -85,B 0,C 180,E1 -11629.217,E2 -11629.217} C_VEL
LIN {X 0,Y 391.691,Z 338.411,A -85,B 0,C 180,E1 -11630.069,E2 -11630.069} C_VEL
LIN {X 0,Y 393.124,Z 318.561,A -85,B 0,C 180,E1 -11633.997,E2 -11633.997} C_VEL
LIN {X 0,Y 393.714,Z 310.294,A -85,B 0,C 180,E1 -11635.649,E2 -11635.649} C_VEL
LIN {X 0,Y 391.095,Z 296.668,A -85,B 0,C 180,E1 -11638.62,E2 -11638.62} C_VEL
LIN {X 0,Y 390.07,Z 291.896,A -85,B 0,C 180,E1 -11639.7,E2 -11639.7} C_VEL
LIN {X 0,Y 390.037,Z 291.903,A -85,B 0,C 180,E1 -11642.72,E2 -11642.72} C_VEL
LIN {X 0,Y 390.036,Z 291.897,A -85,B 0,C 180,E1 -11645.82,E2 -11645.82} C_VEL
LIN {X 0,Y 390.028,Z 291.9,A -85,B 0,C 180,E1 -11649.21,E2 -11649.21} C_VEL
LIN {X 0,Y 390.02,Z 291.901,A -85,B 0,C 180,E1 -11652.37,E2 -11652.37} C_VEL
LIN {X 0,Y 390.028,Z 291.9,A -85,B 0,C 180,E1 -11655.351,E2 -11655.351} C_VEL
LIN {X 0,Y 390.001,Z 291.902,A -85,B 0,C 180,E1 -11658.182,E2 -11658.182} C_VEL
LIN {X 0,Y 390.041,Z 291.902,A -85,B 0,C 180,E1 -11660.901,E2 -11660.901} C_VEL
LIN {X 0,Y 390.051,Z 291.9,A -85,B 0,C 180,E1 -11664.789,E2 -11664.789} C_VEL
LIN {X 0,Y 390,Z 291.904,A -85,B 0,C 180,E1 -11668.493,E2 -11668.493} C_VEL
LIN {X 0,Y 390.055,Z 291.895,A -85,B 0,C 180,E1 -11672.065,E2 -11672.065} C_VEL
LIN {X 0,Y 390.021,Z 291.902,A -85,B 0,C 180,E1 -11675.515,E2 -11675.515} C_VEL
LIN {X 0,Y 390.027,Z 291.903,A -85,B 0,C 180,E1 -11678.876,E2 -11678.876} C_VEL
LIN {X 0,Y 390.086,Z 291.892,A -85,B 0,C 180,E1 -11682.164,E2 -11682.164} C_VEL
LIN {X 0,Y 390.115,Z 291.891,A -85,B 0,C 180,E1 -11685.391,E2 -11685.391} C_VEL
LIN {X 0,Y 390.122,Z 291.888,A -85,B 0,C 180,E1 -11688.57,E2 -11688.57} C_VEL
LIN {X 0,Y 390.28,Z 291.869,A -85,B 0,C 180,E1 -11692.031,E2 -11692.031} C_VEL
LIN {X 0,Y 390.191,Z 291.881,A -85,B 0,C 180,E1 -11694.833,E2 -11694.833} C_VEL
LIN {X 0,Y 390.385,Z 291.857,A -85,B 0,C 180,E1 -11697.936,E2 -11697.936} C_VEL
LIN {X 0,Y 390.516,Z 291.84,A -85,B 0,C 180,E1 -11699.999,E2 -11699.999} C_VEL
LIN {X 0,Y 390.276,Z 291.871,A -85,B 0,C 180,E1 -11703.096,E2 -11703.096} C_VEL
LIN {X 0,Y 390.264,Z 291.87,A -85,B 0,C 180,E1 -11706.712,E2 -11706.712} C_VEL
LIN {X 0,Y 390.177,Z 291.885,A -85,B 0,C 180,E1 -11709.329,E2 -11709.329} C_VEL
LIN {X 0,Y 390.149,Z 291.885,A -85,B 0,C 180,E1 -11712.483,E2 -11712.483} C_VEL
LIN {X 0,Y 390.11,Z 291.892,A -85,B 0,C 180,E1 -11715.677,E2 -11715.677} C_VEL
LIN {X 0,Y 390.071,Z 291.895,A -85,B 0,C 180,E1 -11718.923,E2 -11718.923} C_VEL
LIN {X 0,Y 390.012,Z 291.904,A -85,B 0,C 180,E1 -11722.235,E2 -11722.235} C_VEL
LIN {X 0,Y 390.094,Z 291.894,A -85,B 0,C 180,E1 -11725.744,E2 -11725.744} C_VEL
LIN {X 0,Y 390.04,Z 291.899,A -85,B 0,C 180,E1 -11729.11,E2 -11729.11} C_VEL
LIN {X 0,Y 390.021,Z 291.901,A -85,B 0,C 180,E1 -11732.723,E2 -11732.723} C_VEL
LIN {X 0,Y 390.036,Z 291.901,A -85,B 0,C 180,E1 -11735.826,E2 -11735.826} C_VEL
LIN {X 0,Y 390.055,Z 291.897,A -85,B 0,C 180,E1 -11739.22,E2 -11739.22} C_VEL
LIN {X 0,Y 390.038,Z 291.902,A -85,B 0,C 180,E1 -11742.377,E2 -11742.377} C_VEL
LIN {X 0,Y 390.084,Z 291.895,A -85,B 0,C 180,E1 -11746.109,E2 -11746.109} C_VEL
LIN {X 0,Y 390.069,Z 291.895,A -85,B 0,C 180,E1 -11749.176,E2 -11749.176} C_VEL
LIN {X 0,Y 390.036,Z 291.903,A -85,B 0,C 180,E1 -11752.45,E2 -11752.45} C_VEL
LIN {X 0,Y 390.059,Z 291.898,A -85,B 0,C 180,E1 -11756.046,E2 -11756.046} C_VEL
LIN {X 0,Y 390.038,Z 291.9,A -85,B 0,C 180,E1 -11759.87,E2 -11759.87} C_VEL
LIN {X 0,Y 390.107,Z 291.89,A -85,B 0,C 180,E1 -11763.232,E2 -11763.232} C_VEL
LIN {X 0,Y 390.101,Z 291.893,A -85,B 0,C 180,E1 -11766.751,E2 -11766.751} C_VEL
LIN {X 0,Y 390.1,Z 291.892,A -85,B 0,C 180,E1 -11769.983,E2 -11769.983} C_VEL
LIN {X 0,Y 390.135,Z 291.886,A -85,B 0,C 180,E1 -11773.248,E2 -11773.248} C_VEL
LIN {X 0,Y 390.192,Z 291.883,A -85,B 0,C 180,E1 -11776.561,E2 -11776.561} C_VEL
LIN {X 0,Y 390.203,Z 291.882,A -85,B 0,C 180,E1 -11780.67,E2 -11780.67} C_VEL
LIN {X 0,Y 390.317,Z 291.868,A -85,B 0,C 180,E1 -11782.758,E2 -11782.758} C_VEL
LIN {X 0,Y 390.224,Z 291.879,A -85,B 0,C 180,E1 -11784.832,E2 -11784.832} C_VEL
LIN {X 0,Y 390.417,Z 291.851,A -85,B 0,C 180,E1 -11787.935,E2 -11787.935} C_VEL
LIN {X 0,Y 390.547,Z 291.835,A -85,B 0,C 180,E1 -11789.998,E2 -11789.998} C_VEL
LIN {X 0,Y 390.312,Z 291.866,A -85,B 0,C 180,E1 -11793.095,E2 -11793.095} C_VEL
LIN {X 0,Y 390.322,Z 291.864,A -85,B 0,C 180,E1 -11796.2,E2 -11796.2} C_VEL
LIN {X 0,Y 390.309,Z 291.865,A -85,B 0,C 180,E1 -11798.28,E2 -11798.28} C_VEL
LIN {X 0,Y 390.171,Z 291.883,A -85,B 0,C 180,E1 -11802.48,E2 -11802.48} C_VEL
LIN {X 0,Y 390.131,Z 291.886,A -85,B 0,C 180,E1 -11805.674,E2 -11805.674} C_VEL
LIN {X 0,Y 390.109,Z 291.894,A -85,B 0,C 180,E1 -11808.918,E2 -11808.918} C_VEL
LIN {X 0,Y 390.053,Z 291.896,A -85,B 0,C 180,E1 -11812.229,E2 -11812.229} C_VEL
LIN {X 0,Y 390.104,Z 291.889,A -85,B 0,C 180,E1 -11815.74,E2 -11815.74} C_VEL
LIN {X 0,Y 390.048,Z 291.902,A -85,B 0,C 180,E1 -11819.105,E2 -11819.105} C_VEL
LIN {X 0,Y 389.998,Z 291.9,A -85,B 0,C 180,E1 -11820.833,E2 -11820.833} C_VEL
LIN {X 0,Y 389.326,Z 291.988,A -85,B 0,C 180,E1 -11821.695,E2 -11821.695} C_VEL
LIN {X 0,Y 386.474,Z 292.347,A -85,B 0,C 180,E1 -11823.097,E2 -11823.097} C_VEL
LIN {X 0,Y 384.071,Z 292.642,A -85,B 0,C 180,E1 -11824.229,E2 -11824.229} C_VEL
LIN {X 0,Y 383.053,Z 292.773,A -85,B 0,C 180,E1 -11825.105,E2 -11825.105} C_VEL
LIN {X 0,Y 382.976,Z 292.774,A -85,B 0,C 180,E1 -11825.402,E2 -11825.402} C_VEL
LIN {X 0,Y 382.983,Z 292.777,A -85,B 0,C 180,E1 -11828.596,E2 -11828.596} C_VEL
LIN {X 0,Y 383.089,Z 292.955,A -85,B 0,C 180,E1 -11830.717,E2 -11830.717} C_VEL
LIN {X 0,Y 383.786,Z 296.655,A -85,B 0,C 180,E1 -11831.672,E2 -11831.672} C_VEL
LIN {X 0,Y 387.902,Z 309.831,A -85,B 0,C 180,E1 -11832.166,E2 -11832.166} C_VEL
LIN {X 0,Y 389.527,Z 317.96,A -85,B 0,C 180,E1 -11832.419,E2 -11832.419} C_VEL
LIN {X 0,Y 387.842,Z 404.756,A -85,B 0,C 180,E1 -11834.248,E2 -11834.248} C_VEL
LIN {X 0,Y 387.491,Z 418.308,A -85,B 0,C 180,E1 -11834.751,E2 -11834.751} C_VEL
LIN {X 0,Y 386.901,Z 431.162,A -85,B 0,C 180,E1 -11835.444,E2 -11835.444} C_VEL
LIN {X 0,Y 386.289,Z 442.492,A -85,B 0,C 180,E1 -11836.263,E2 -11836.263} C_VEL
LIN {X 0,Y 385.551,Z 453.52,A -85,B 0,C 180,E1 -11837.271,E2 -11837.271} C_VEL
LIN {X 0,Y 384.819,Z 464.107,A -85,B 0,C 180,E1 -11838.476,E2 -11838.476} C_VEL
LIN {X 0,Y 384.073,Z 473.669,A -85,B 0,C 180,E1 -11839.833,E2 -11839.833} C_VEL
LIN {X 0,Y 383.384,Z 482.848,A -85,B 0,C 180,E1 -11841.445,E2 -11841.445} C_VEL
LIN {X 0,Y 382.832,Z 490.08,A -85,B 0,C 180,E1 -11843.044,E2 -11843.044} C_VEL
LIN {X 0,Y 382.398,Z 495.787,A -85,B 0,C 180,E1 -11844.625,E2 -11844.625} C_VEL
LIN {X 0,Y 382.071,Z 501.005,A -85,B 0,C 180,E1 -11846.508,E2 -11846.508} C_VEL
LIN {X 0,Y 381.865,Z 503.735,A -85,B 0,C 180,E1 -11847.832,E2 -11847.832} C_VEL
LIN {X 0,Y 381.685,Z 505.535,A -85,B 0,C 180,E1 -11848.965,E2 -11848.965} C_VEL
LIN {X 0,Y 381.612,Z 506.887,A -85,B 0,C 180,E1 -11850.183,E2 -11850.183} C_VEL
LIN {X 0,Y 381.599,Z 507.91,A -85,B 0,C 180,E1 -11852.118,E2 -11852.118} C_VEL
LIN {X 0,Y 381.651,Z 507.689,A -85,B 0,C 180,E1 -11853.772,E2 -11853.772} C_VEL
LIN {X 0,Y 381.784,Z 506.934,A -85,B 0,C 180,E1 -11854.952,E2 -11854.952} C_VEL
LIN {X 0,Y 382.078,Z 504.533,A -85,B 0,C 180,E1 -11856.865,E2 -11856.865} C_VEL
LIN {X 0,Y 382.398,Z 501.519,A -85,B 0,C 180,E1 -11858.434,E2 -11858.434} C_VEL
LIN {X 0,Y 382.841,Z 497.02,A -85,B 0,C 180,E1 -11860.147,E2 -11860.147} C_VEL
LIN {X 0,Y 383.495,Z 491.164,A -85,B 0,C 180,E1 -11861.848,E2 -11861.848} C_VEL
LIN {X 0,Y 384.268,Z 483.759,A -85,B 0,C 180,E1 -11863.532,E2 -11863.532} C_VEL
LIN {X 0,Y 385.098,Z 475.938,A -85,B 0,C 180,E1 -11864.954,E2 -11864.954} C_VEL
LIN {X 0,Y 386.124,Z 465.778,A -85,B 0,C 180,E1 -11866.448,E2 -11866.448} C_VEL
LIN {X 0,Y 387.148,Z 455.293,A -85,B 0,C 180,E1 -11867.667,E2 -11867.667} C_VEL
LIN {X 0,Y 388.063,Z 443.372,A -85,B 0,C 180,E1 -11868.774,E2 -11868.774} C_VEL
LIN {X 0,Y 388.896,Z 431.034,A -85,B 0,C 180,E1 -11869.655,E2 -11869.655} C_VEL
LIN {X 0,Y 389.54,Z 417.594,A -85,B 0,C 180,E1 -11870.361,E2 -11870.361} C_VEL
LIN {X 0,Y 390.01,Z 405.248,A -85,B 0,C 180,E1 -11870.797,E2 -11870.797} C_VEL
LIN {X 0,Y 392.132,Z 318.274,A -85,B 0,C 180,E1 -11872.725,E2 -11872.725} C_VEL
LIN {X 0,Y 390.837,Z 312.837,A -85,B 0,C 180,E1 -11872.948,E2 -11872.948} C_VEL
LIN {X 0,Y 385.116,Z 299.237,A -85,B 0,C 180,E1 -11873.714,E2 -11873.714} C_VEL
LIN {X 0,Y 384.515,Z 297.57,A -85,B 0,C 180,E1 -11873.836,E2 -11873.836} C_VEL
LIN {X 0,Y 383.113,Z 292.77,A -85,B 0,C 180,E1 -11874.936,E2 -11874.936} C_VEL
LIN {X 0,Y 383.336,Z 292.739,A -85,B 0,C 180,E1 -11877.899,E2 -11877.899} C_VEL
LIN {X 0,Y 383.466,Z 292.718,A -85,B 0,C 180,E1 -11880.001,E2 -11880.001} C_VEL
LIN {X 0,Y 383.204,Z 292.753,A -85,B 0,C 180,E1 -11883.155,E2 -11883.155} C_VEL
LIN {X 0,Y 383.23,Z 292.747,A -85,B 0,C 180,E1 -11886.318,E2 -11886.318} C_VEL
LIN {X 0,Y 383.104,Z 292.764,A -85,B 0,C 180,E1 -11889.504,E2 -11889.504} C_VEL
LIN {X 0,Y 383.094,Z 292.763,A -85,B 0,C 180,E1 -11892.718,E2 -11892.718} C_VEL
LIN {X 0,Y 383.033,Z 292.77,A -85,B 0,C 180,E1 -11895.976,E2 -11895.976} C_VEL
LIN {X 0,Y 383.005,Z 292.775,A -85,B 0,C 180,E1 -11899.287,E2 -11899.287} C_VEL
LIN {X 0,Y 382.952,Z 292.781,A -85,B 0,C 180,E1 -11902.669,E2 -11902.669} C_VEL
LIN {X 0,Y 383.039,Z 292.766,A -85,B 0,C 180,E1 -11906.127,E2 -11906.127} C_VEL
LIN {X 0,Y 382.952,Z 292.783,A -85,B 0,C 180,E1 -11909.704,E2 -11909.704} C_VEL
LIN {X 0,Y 382.966,Z 292.78,A -85,B 0,C 180,E1 -11913.405,E2 -11913.405} C_VEL
LIN {X 0,Y 382.999,Z 292.775,A -85,B 0,C 180,E1 -11916.168,E2 -11916.168} C_VEL
LIN {X 0,Y 382.988,Z 292.775,A -85,B 0,C 180,E1 -11919.961,E2 -11919.961} C_VEL
LIN {X 0,Y 382.978,Z 292.776,A -85,B 0,C 180,E1 -11922.783,E2 -11922.783} C_VEL
LIN {X 0,Y 382.971,Z 292.781,A -85,B 0,C 180,E1 -11925.793,E2 -11925.793} C_VEL
LIN {X 0,Y 382.964,Z 292.781,A -85,B 0,C 180,E1 -11928.801,E2 -11928.801} C_VEL
LIN {X 0,Y 382.977,Z 292.778,A -85,B 0,C 180,E1 -11932.101,E2 -11932.101} C_VEL
LIN {X 0,Y 383.001,Z 292.782,A -85,B 0,C 180,E1 -11935.336,E2 -11935.336} C_VEL
LIN {X 0,Y 382.968,Z 292.791,A -85,B 0,C 180,E1 -11939.086,E2 -11939.086} C_VEL
LIN {X 0,Y 383.028,Z 292.976,A -85,B 0,C 180,E1 -11939.896,E2 -11939.896} C_VEL
LIN {X 0,Y 385.988,Z 305.2,A -85,B 0,C 180,E1 -11942.634,E2 -11942.634} C_VEL
LIN {X 0,Y 387.129,Z 311.154,A -85,B 0,C 180,E1 -11943.9,E2 -11943.9} C_VEL
LIN {X 0,Y 386.497,Z 321.534,A -85,B 0,C 180,E1 -11945.886,E2 -11945.886} C_VEL
LIN {X 0,Y 385.557,Z 334.507,A -85,B 0,C 180,E1 -11948.34,E2 -11948.34} C_VEL
LIN {X 0,Y 389.1,Z 354.166,A -85,B 0,C 180,E1 -11949.076,E2 -11949.076} C_VEL
LIN {X 0,Y 391.21,Z 371.517,A -85,B 0,C 180,E1 -11949.631,E2 -11949.631} C_VEL
LIN {X 0,Y 389.398,Z 446.113,A -85,B 0,C 180,E1 -11951.285,E2 -11951.285} C_VEL
LIN {X 0,Y 388.62,Z 459.859,A -85,B 0,C 180,E1 -11951.792,E2 -11951.792} C_VEL
LIN {X 0,Y 387.716,Z 472.316,A -85,B 0,C 180,E1 -11952.465,E2 -11952.465} C_VEL
LIN {X 0,Y 386.636,Z 484.77,A -85,B 0,C 180,E1 -11953.367,E2 -11953.367} C_VEL
LIN {X 0,Y 385.633,Z 496.005,A -85,B 0,C 180,E1 -11954.41,E2 -11954.41} C_VEL
LIN {X 0,Y 384.607,Z 506.979,A -85,B 0,C 180,E1 -11955.696,E2 -11955.696} C_VEL
LIN {X 0,Y 383.77,Z 516.268,A -85,B 0,C 180,E1 -11957.039,E2 -11957.039} C_VEL
LIN {X 0,Y 382.853,Z 525.182,A -85,B 0,C 180,E1 -11958.622,E2 -11958.622} C_VEL
LIN {X 0,Y 382.27,Z 532.323,A -85,B 0,C 180,E1 -11960.211,E2 -11960.211} C_VEL
LIN {X 0,Y 381.888,Z 538.928,A -85,B 0,C 180,E1 -11962.069,E2 -11962.069} C_VEL
LIN {X 0,Y 381.674,Z 543.846,A -85,B 0,C 180,E1 -11963.903,E2 -11963.903} C_VEL
LIN {X 0,Y 381.654,Z 547.37,A -85,B 0,C 180,E1 -11965.778,E2 -11965.778} C_VEL
LIN {X 0,Y 381.627,Z 548.758,A -85,B 0,C 180,E1 -11966.835,E2 -11966.835} C_VEL
LIN {X 0,Y 381.729,Z 549.739,A -85,B 0,C 180,E1 -11967.892,E2 -11967.892} C_VEL
LIN {X 0,Y 381.722,Z 550.252,A -85,B 0,C 180,E1 -11968.947,E2 -11968.947} C_VEL
LIN {X 0,Y 381.731,Z 550.349,A -85,B 0,C 180,E1 -11970.002,E2 -11970.002} C_VEL
LIN {X 0,Y 381.732,Z 550.041,A -85,B 0,C 180,E1 -11971.056,E2 -11971.056} C_VEL
LIN {X 0,Y 381.771,Z 549.318,A -85,B 0,C 180,E1 -11972.111,E2 -11972.111} C_VEL
LIN {X 0,Y 381.665,Z 548.114,A -85,B 0,C 180,E1 -11973.168,E2 -11973.168} C_VEL
LIN {X 0,Y 381.733,Z 545.518,A -85,B 0,C 180,E1 -11974.754,E2 -11974.754} C_VEL
LIN {X 0,Y 381.769,Z 541.844,A -85,B 0,C 180,E1 -11976.343,E2 -11976.343} C_VEL
LIN {X 0,Y 381.894,Z 537.002,A -85,B 0,C 180,E1 -11977.934,E2 -11977.934} C_VEL
LIN {X 0,Y 382.18,Z 530.851,A -85,B 0,C 180,E1 -11979.527,E2 -11979.527} C_VEL
LIN {X 0,Y 382.645,Z 523.172,A -85,B 0,C 180,E1 -11981.12,E2 -11981.12} C_VEL
LIN {X 0,Y 383.254,Z 515.326,A -85,B 0,C 180,E1 -11982.443,E2 -11982.443} C_VEL
LIN {X 0,Y 384.008,Z 505.732,A -85,B 0,C 180,E1 -11983.764,E2 -11983.764} C_VEL
LIN {X 0,Y 384.746,Z 495.08,A -85,B 0,C 180,E1 -11984.953,E2 -11984.953} C_VEL
LIN {X 0,Y 385.605,Z 483.253,A -85,B 0,C 180,E1 -11986.002,E2 -11986.002} C_VEL
LIN {X 0,Y 386.38,Z 470.666,A -85,B 0,C 180,E1 -11986.852,E2 -11986.852} C_VEL
LIN {X 0,Y 387.188,Z 457.604,A -85,B 0,C 180,E1 -11987.496,E2 -11987.496} C_VEL
LIN {X 0,Y 387.67,Z 444.652,A -85,B 0,C 180,E1 -11987.916,E2 -11987.916} C_VEL
LIN {X 0,Y 388.871,Z 369.555,A -85,B 0,C 180,E1 -11989.495,E2 -11989.495} C_VEL
LIN {X 0,Y 384.729,Z 338.113,A -85,B 0,C 180,E1 -11990.378,E2 -11990.378} C_VEL
LIN {X 0,Y 386.144,Z 319.603,A -85,B 0,C 180,E1 -11994.104,E2 -11994.104} C_VEL
LIN {X 0,Y 386.753,Z 312.403,A -85,B 0,C 180,E1 -11995.567,E2 -11995.567} C_VEL
LIN {X 0,Y 385.604,Z 305.362,A -85,B 0,C 180,E1 -11997.106,E2 -11997.106} C_VEL
LIN {X 0,Y 383.026,Z 292.775,A -85,B 0,C 180,E1 -11999.99,E2 -11999.99} C_VEL
LIN {X 0,Y 382.995,Z 292.775,A -85,B 0,C 180,E1 -12003.4,E2 -12003.4} C_VEL
LIN {X 0,Y 383.015,Z 292.773,A -85,B 0,C 180,E1 -12006.16,E2 -12006.16} C_VEL
LIN {X 0,Y 382.977,Z 292.777,A -85,B 0,C 180,E1 -12009.579,E2 -12009.579} C_VEL
LIN {X 0,Y 382.997,Z 292.78,A -85,B 0,C 180,E1 -12012.777,E2 -12012.777} C_VEL
LIN {X 0,Y 382.977,Z 292.777,A -85,B 0,C 180,E1 -12015.786,E2 -12015.786} C_VEL
LIN {X 0,Y 382.948,Z 292.786,A -85,B 0,C 180,E1 -12018.799,E2 -12018.799} C_VEL
LIN {X 0,Y 382.977,Z 292.777,A -85,B 0,C 180,E1 -12022.096,E2 -12022.096} C_VEL
LIN {X 0,Y 382.994,Z 292.777,A -85,B 0,C 180,E1 -12025.329,E2 -12025.329} C_VEL
LIN {X 0,Y 382.961,Z 292.783,A -85,B 0,C 180,E1 -12029.079,E2 -12029.079} C_VEL
LIN {X 0,Y 382.999,Z 292.777,A -85,B 0,C 180,E1 -12032.693,E2 -12032.693} C_VEL
LIN {X 0,Y 382.989,Z 292.776,A -85,B 0,C 180,E1 -12036.189,E2 -12036.189} C_VEL
LIN {X 0,Y 383.016,Z 292.774,A -85,B 0,C 180,E1 -12039.596,E2 -12039.596} C_VEL
LIN {X 0,Y 383.071,Z 292.769,A -85,B 0,C 180,E1 -12042.929,E2 -12042.929} C_VEL
LIN {X 0,Y 383.1,Z 292.762,A -85,B 0,C 180,E1 -12046.463,E2 -12046.463} C_VEL
LIN {X 0,Y 383.124,Z 292.759,A -85,B 0,C 180,E1 -12050.497,E2 -12050.497} C_VEL
LIN {X 0,Y 383.226,Z 292.747,A -85,B 0,C 180,E1 -12052.624,E2 -12052.624} C_VEL
LIN {X 0,Y 383.163,Z 292.755,A -85,B 0,C 180,E1 -12054.737,E2 -12054.737} C_VEL
LIN {X 0,Y 383.353,Z 292.733,A -85,B 0,C 180,E1 -12057.898,E2 -12057.898} C_VEL
LIN {X 0,Y 383.486,Z 292.716,A -85,B 0,C 180,E1 -12059.999,E2 -12059.999} C_VEL
LIN {X 0,Y 383.212,Z 292.752,A -85,B 0,C 180,E1 -12063.153,E2 -12063.153} C_VEL
LIN {X 0,Y 383.223,Z 292.747,A -85,B 0,C 180,E1 -12066.705,E2 -12066.705} C_VEL
LIN {X 0,Y 383.124,Z 292.763,A -85,B 0,C 180,E1 -12069.502,E2 -12069.502} C_VEL
LIN {X 0,Y 383.113,Z 292.761,A -85,B 0,C 180,E1 -12072.716,E2 -12072.716} C_VEL
LIN {X 0,Y 383.051,Z 292.771,A -85,B 0,C 180,E1 -12075.974,E2 -12075.974} C_VEL
LIN {X 0,Y 383.023,Z 292.775,A -85,B 0,C 180,E1 -12079.285,E2 -12079.285} C_VEL
LIN {X 0,Y 382.97,Z 292.779,A -85,B 0,C 180,E1 -12082.667,E2 -12082.667} C_VEL
LIN {X 0,Y 383.056,Z 292.771,A -85,B 0,C 180,E1 -12086.124,E2 -12086.124} C_VEL
LIN {X 0,Y 383.019,Z 292.774,A -85,B 0,C 180,E1 -12088.494,E2 -12088.494} C_VEL
LIN {X 0,Y 382.988,Z 292.78,A -85,B 0,C 180,E1 -12092.151,E2 -12092.151} C_VEL
LIN {X 0,Y 382.998,Z 292.776,A -85,B 0,C 180,E1 -12094.669,E2 -12094.669} C_VEL
LIN {X 0,Y 382.984,Z 292.78,A -85,B 0,C 180,E1 -12097.905,E2 -12097.905} C_VEL
LIN {X 0,Y 382.986,Z 292.778,A -85,B 0,C 180,E1 -12101.346,E2 -12101.346} C_VEL
LIN {X 0,Y 382.989,Z 292.78,A -85,B 0,C 180,E1 -12104.306,E2 -12104.306} C_VEL
LIN {X 0,Y 383.062,Z 292.767,A -85,B 0,C 180,E1 -12107.25,E2 -12107.25} C_VEL
LIN {X 0,Y 383.01,Z 292.778,A -85,B 0,C 180,E1 -12110.414,E2 -12110.414} C_VEL
LIN {X 0,Y 383.016,Z 292.776,A -85,B 0,C 180,E1 -12114.046,E2 -12114.046} C_VEL
LIN {X 0,Y 382.977,Z 292.779,A -85,B 0,C 180,E1 -12117.579,E2 -12117.579} C_VEL
LIN {X 0,Y 382.984,Z 292.78,A -85,B 0,C 180,E1 -12120.301,E2 -12120.301} C_VEL
LIN {X 0,Y 383.074,Z 292.768,A -85,B 0,C 180,E1 -12124.021,E2 -12124.021} C_VEL
LIN {X 0,Y 383.003,Z 292.774,A -85,B 0,C 180,E1 -12127.336,E2 -12127.336} C_VEL
LIN {X 0,Y 383.056,Z 292.771,A -85,B 0,C 180,E1 -12130.716,E2 -12130.716} C_VEL
LIN {X 0,Y 383.078,Z 292.767,A -85,B 0,C 180,E1 -12134.026,E2 -12134.026} C_VEL
LIN {X 0,Y 383.134,Z 292.758,A -85,B 0,C 180,E1 -12137.283,E2 -12137.283} C_VEL
LIN {X 0,Y 383.149,Z 292.759,A -85,B 0,C 180,E1 -12140.497,E2 -12140.497} C_VEL
LIN {X 0,Y 383.271,Z 292.745,A -85,B 0,C 180,E1 -12142.624,E2 -12142.624} C_VEL
LIN {X 0,Y 383.196,Z 292.755,A -85,B 0,C 180,E1 -12144.737,E2 -12144.737} C_VEL
LIN {X 0,Y 383.385,Z 292.727,A -85,B 0,C 180,E1 -12147.897,E2 -12147.897} C_VEL
LIN {X 0,Y 383.517,Z 292.711,A -85,B 0,C 180,E1 -12149.998,E2 -12149.998} C_VEL
LIN {X 0,Y 383.248,Z 292.745,A -85,B 0,C 180,E1 -12153.152,E2 -12153.152} C_VEL
LIN {X 0,Y 383.279,Z 292.741,A -85,B 0,C 180,E1 -12156.314,E2 -12156.314} C_VEL
LIN {X 0,Y 383.255,Z 292.745,A -85,B 0,C 180,E1 -12158.433,E2 -12158.433} C_VEL
LIN {X 0,Y 383.1,Z 292.762,A -85,B 0,C 180,E1 -12161.639,E2 -12161.639} C_VEL
LIN {X 0,Y 383.104,Z 292.766,A -85,B 0,C 180,E1 -12164.879,E2 -12164.879} C_VEL
LIN {X 0,Y 383.084,Z 292.764,A -85,B 0,C 180,E1 -12168.169,E2 -12168.169} C_VEL
LIN {X 0,Y 383.01,Z 292.774,A -85,B 0,C 180,E1 -12171.526,E2 -12171.526} C_VEL
LIN {X 0,Y 383.038,Z 292.774,A -85,B 0,C 180,E1 -12174.957,E2 -12174.957} C_VEL
LIN {X 0,Y 383.032,Z 292.771,A -85,B 0,C 180,E1 -12178.488,E2 -12178.488} C_VEL
LIN {X 0,Y 382.993,Z 292.774,A -85,B 0,C 180,E1 -12182.146,E2 -12182.146} C_VEL
LIN {X 0,Y 382.976,Z 292.774,A -85,B 0,C 180,E1 -12185.402,E2 -12185.402} C_VEL
LIN {X 0,Y 382.332,Z 292.857,A -85,B 0,C 180,E1 -12186.28,E2 -12186.28} C_VEL
LIN {X 0,Y 379.509,Z 293.212,A -85,B 0,C 180,E1 -12187.707,E2 -12187.707} C_VEL
LIN {X 0,Y 377.107,Z 293.513,A -85,B 0,C 180,E1 -12188.862,E2 -12188.862} C_VEL
LIN {X 0,Y 376.071,Z 293.642,A -85,B 0,C 180,E1 -12189.754,E2 -12189.754} C_VEL
LIN {X 0,Y 375.986,Z 293.652,A -85,B 0,C 180,E1 -12190.056,E2 -12190.056} C_VEL
LIN {X 0,Y 376.006,Z 293.759,A -85,B 0,C 180,E1 -12190.483,E2 -12190.483} C_VEL
LIN {X 0,Y 376.706,Z 297.268,A -85,B 0,C 180,E1 -12191.354,E2 -12191.354} C_VEL
LIN {X 0,Y 381.299,Z 311.739,A -85,B 0,C 180,E1 -12191.904,E2 -12191.904} C_VEL
LIN {X 0,Y 382.723,Z 319.726,A -85,B 0,C 180,E1 -12192.15,E2 -12192.15} C_VEL
LIN {X 0,Y 380.973,Z 405.229,A -85,B 0,C 180,E1 -12193.992,E2 -12193.992} C_VEL
LIN {X 0,Y 380.575,Z 419.014,A -85,B 0,C 180,E1 -12194.515,E2 -12194.515} C_VEL
LIN {X 0,Y 380.02,Z 431.3,A -85,B 0,C 180,E1 -12195.191,E2 -12195.191} C_VEL
LIN {X 0,Y 379.298,Z 443.782,A -85,B 0,C 180,E1 -12196.117,E2 -12196.117} C_VEL
LIN {X 0,Y 378.54,Z 454.802,A -85,B 0,C 180,E1 -12197.159,E2 -12197.159} C_VEL
LIN {X 0,Y 377.832,Z 464.912,A -85,B 0,C 180,E1 -12198.351,E2 -12198.351} C_VEL
LIN {X 0,Y 376.993,Z 475.071,A -85,B 0,C 180,E1 -12199.838,E2 -12199.838} C_VEL
LIN {X 0,Y 376.398,Z 482.645,A -85,B 0,C 180,E1 -12201.2,E2 -12201.2} C_VEL
LIN {X 0,Y 375.799,Z 490.337,A -85,B 0,C 180,E1 -12202.907,E2 -12202.907} C_VEL
LIN {X 0,Y 375.358,Z 496.085,A -85,B 0,C 180,E1 -12204.52,E2 -12204.52} C_VEL
LIN {X 0,Y 375.012,Z 501.333,A -85,B 0,C 180,E1 -12206.438,E2 -12206.438} C_VEL
LIN {X 0,Y 374.682,Z 505.006,A -85,B 0,C 180,E1 -12208.319,E2 -12208.319} C_VEL
LIN {X 0,Y 374.564,Z 506.747,A -85,B 0,C 180,E1 -12209.654,E2 -12209.654} C_VEL
LIN {X 0,Y 374.512,Z 507.765,A -85,B 0,C 180,E1 -12210.797,E2 -12210.797} C_VEL
LIN {X 0,Y 374.513,Z 508.285,A -85,B 0,C 180,E1 -12212.022,E2 -12212.022} C_VEL
LIN {X 0,Y 374.542,Z 508.318,A -85,B 0,C 180,E1 -12213.235,E2 -12213.235} C_VEL
LIN {X 0,Y 374.639,Z 507.802,A -85,B 0,C 180,E1 -12214.44,E2 -12214.44} C_VEL
LIN {X 0,Y 374.79,Z 506.785,A -85,B 0,C 180,E1 -12215.636,E2 -12215.636} C_VEL
LIN {X 0,Y 375.142,Z 504.31,A -85,B 0,C 180,E1 -12217.416,E2 -12217.416} C_VEL
LIN {X 0,Y 375.538,Z 500.288,A -85,B 0,C 180,E1 -12219.325,E2 -12219.325} C_VEL
LIN {X 0,Y 376.052,Z 495.755,A -85,B 0,C 180,E1 -12220.91,E2 -12220.91} C_VEL
LIN {X 0,Y 376.778,Z 489.412,A -85,B 0,C 180,E1 -12222.636,E2 -12222.636} C_VEL
LIN {X 0,Y 377.704,Z 481.441,A -85,B 0,C 180,E1 -12224.348,E2 -12224.348} C_VEL
LIN {X 0,Y 378.635,Z 472.962,A -85,B 0,C 180,E1 -12225.798,E2 -12225.798} C_VEL
LIN {X 0,Y 379.675,Z 463.106,A -85,B 0,C 180,E1 -12227.167,E2 -12227.167} C_VEL
LIN {X 0,Y 380.789,Z 451.772,A -85,B 0,C 180,E1 -12228.422,E2 -12228.422} C_VEL
LIN {X 0,Y 381.647,Z 440.738,A -85,B 0,C 180,E1 -12229.389,E2 -12229.389} C_VEL
LIN {X 0,Y 382.468,Z 428.6,A -85,B 0,C 180,E1 -12230.214,E2 -12230.214} C_VEL
LIN {X 0,Y 383.029,Z 416.412,A -85,B 0,C 180,E1 -12230.829,E2 -12230.829} C_VEL
LIN {X 0,Y 383.527,Z 402.848,A -85,B 0,C 180,E1 -12231.273,E2 -12231.273} C_VEL
LIN {X 0,Y 385.81,Z 320.005,A -85,B 0,C 180,E1 -12233.135,E2 -12233.135} C_VEL
LIN {X 0,Y 384.649,Z 315.231,A -85,B 0,C 180,E1 -12233.345,E2 -12233.345} C_VEL
LIN {X 0,Y 378.654,Z 300.973,A -85,B 0,C 180,E1 -12234.18,E2 -12234.18} C_VEL
LIN {X 0,Y 377.423,Z 298.246,A -85,B 0,C 180,E1 -12234.364,E2 -12234.364} C_VEL
LIN {X 0,Y 376.041,Z 293.65,A -85,B 0,C 180,E1 -12235.445,E2 -12235.445} C_VEL
LIN {X 0,Y 376.302,Z 293.615,A -85,B 0,C 180,E1 -12237.86,E2 -12237.86} C_VEL
LIN {X 0,Y 376.436,Z 293.594,A -85,B 0,C 180,E1 -12240.001,E2 -12240.001} C_VEL
LIN {X 0,Y 376.142,Z 293.633,A -85,B 0,C 180,E1 -12243.214,E2 -12243.214} C_VEL
LIN {X 0,Y 376.189,Z 293.624,A -85,B 0,C 180,E1 -12246.436,E2 -12246.436} C_VEL
LIN {X 0,Y 376.072,Z 293.639,A -85,B 0,C 180,E1 -12249.683,E2 -12249.683} C_VEL
LIN {X 0,Y 376.044,Z 293.643,A -85,B 0,C 180,E1 -12253.66,E2 -12253.66} C_VEL
LIN {X 0,Y 375.986,Z 293.646,A -85,B 0,C 180,E1 -12257.403,E2 -12257.403} C_VEL
LIN {X 0,Y 375.936,Z 293.652,A -85,B 0,C 180,E1 -12260.835,E2 -12260.835} C_VEL
LIN {X 0,Y 375.948,Z 293.653,A -85,B 0,C 180,E1 -12264.285,E2 -12264.285} C_VEL
LIN {X 0,Y 375.98,Z 293.647,A -85,B 0,C 180,E1 -12266.656,E2 -12266.656} C_VEL
LIN {X 0,Y 375.926,Z 293.657,A -85,B 0,C 180,E1 -12270.317,E2 -12270.317} C_VEL
LIN {X 0,Y 375.925,Z 293.653,A -85,B 0,C 180,E1 -12274.116,E2 -12274.116} C_VEL
LIN {X 0,Y 375.922,Z 293.657,A -85,B 0,C 180,E1 -12276.745,E2 -12276.745} C_VEL
LIN {X 0,Y 375.967,Z 293.65,A -85,B 0,C 180,E1 -12279.976,E2 -12279.976} C_VEL
LIN {X 0,Y 375.903,Z 293.66,A -85,B 0,C 180,E1 -12283.771,E2 -12283.771} C_VEL
LIN {X 0,Y 375.91,Z 293.659,A -85,B 0,C 180,E1 -12286.815,E2 -12286.815} C_VEL
LIN {X 0,Y 375.936,Z 293.655,A -85,B 0,C 180,E1 -12290.541,E2 -12290.541} C_VEL
LIN {X 0,Y 375.944,Z 293.658,A -85,B 0,C 180,E1 -12293.5,E2 -12293.5} C_VEL
LIN {X 0,Y 375.943,Z 293.662,A -85,B 0,C 180,E1 -12295.893,E2 -12295.893} C_VEL
LIN {X 0,Y 375.978,Z 293.841,A -85,B 0,C 180,E1 -12299.416,E2 -12299.416} C_VEL
LIN {X 0,Y 378.519,Z 303.884,A -85,B 0,C 180,E1 -12301.746,E2 -12301.746} C_VEL
LIN {X 0,Y 380.286,Z 312.637,A -85,B 0,C 180,E1 -12303.675,E2 -12303.675} C_VEL
LIN {X 0,Y 379.946,Z 319.391,A -85,B 0,C 180,E1 -12305.01,E2 -12305.01} C_VEL
LIN {X 0,Y 378.821,Z 334.004,A -85,B 0,C 180,E1 -12307.82,E2 -12307.82} C_VEL
LIN {X 0,Y 382.371,Z 353.505,A -85,B 0,C 180,E1 -12308.588,E2 -12308.588} C_VEL
LIN {X 0,Y 384.724,Z 371.791,A -85,B 0,C 180,E1 -12309.205,E2 -12309.205} C_VEL
LIN {X 0,Y 382.818,Z 445.819,A -85,B 0,C 180,E1 -12310.881,E2 -12310.881} C_VEL
LIN {X 0,Y 382.033,Z 459.417,A -85,B 0,C 180,E1 -12311.398,E2 -12311.398} C_VEL
LIN {X 0,Y 381.126,Z 470.805,A -85,B 0,C 180,E1 -12312.012,E2 -12312.012} C_VEL
LIN {X 0,Y 380.028,Z 483.434,A -85,B 0,C 180,E1 -12312.931,E2 -12312.931} C_VEL
LIN {X 0,Y 378.941,Z 494.785,A -85,B 0,C 180,E1 -12313.989,E2 -12313.989} C_VEL
LIN {X 0,Y 377.92,Z 504.59,A -85,B 0,C 180,E1 -12315.115,E2 -12315.115} C_VEL
LIN {X 0,Y 376.956,Z 514.506,A -85,B 0,C 180,E1 -12316.526,E2 -12316.526} C_VEL
LIN {X 0,Y 376.06,Z 523.676,A -85,B 0,C 180,E1 -12318.14,E2 -12318.14} C_VEL
LIN {X 0,Y 375.341,Z 531.071,A -85,B 0,C 180,E1 -12319.756,E2 -12319.756} C_VEL
LIN {X 0,Y 374.943,Z 536.988,A -85,B 0,C 180,E1 -12321.378,E2 -12321.378} C_VEL
LIN {X 0,Y 374.72,Z 541.671,A -85,B 0,C 180,E1 -12323,E2 -12323} C_VEL
LIN {X 0,Y 374.567,Z 545.239,A -85,B 0,C 180,E1 -12324.619,E2 -12324.619} C_VEL
LIN {X 0,Y 374.578,Z 547.031,A -85,B 0,C 180,E1 -12325.698,E2 -12325.698} C_VEL
LIN {X 0,Y 374.536,Z 548.406,A -85,B 0,C 180,E1 -12326.775,E2 -12326.775} C_VEL
LIN {X 0,Y 374.629,Z 549.364,A -85,B 0,C 180,E1 -12327.852,E2 -12327.852} C_VEL
LIN {X 0,Y 374.654,Z 549.856,A -85,B 0,C 180,E1 -12328.927,E2 -12328.927} C_VEL
LIN {X 0,Y 374.659,Z 549.938,A -85,B 0,C 180,E1 -12330.002,E2 -12330.002} C_VEL
LIN {X 0,Y 374.664,Z 549.613,A -85,B 0,C 180,E1 -12331.076,E2 -12331.076} C_VEL
LIN {X 0,Y 374.685,Z 548.857,A -85,B 0,C 180,E1 -12332.151,E2 -12332.151} C_VEL
LIN {X 0,Y 374.572,Z 547.629,A -85,B 0,C 180,E1 -12333.228,E2 -12333.228} C_VEL
LIN {X 0,Y 374.663,Z 544.992,A -85,B 0,C 180,E1 -12334.843,E2 -12334.843} C_VEL
LIN {X 0,Y 374.713,Z 541.272,A -85,B 0,C 180,E1 -12336.462,E2 -12336.462} C_VEL
LIN {X 0,Y 374.839,Z 536.377,A -85,B 0,C 180,E1 -12338.085,E2 -12338.085} C_VEL
LIN {X 0,Y 375.134,Z 530.165,A -85,B 0,C 180,E1 -12339.708,E2 -12339.708} C_VEL
LIN {X 0,Y 375.647,Z 522.419,A -85,B 0,C 180,E1 -12341.33,E2 -12341.33} C_VEL
LIN {X 0,Y 376.235,Z 514.472,A -85,B 0,C 180,E1 -12342.679,E2 -12342.679} C_VEL
LIN {X 0,Y 377.04,Z 504.76,A -85,B 0,C 180,E1 -12344.024,E2 -12344.024} C_VEL
LIN {X 0,Y 377.813,Z 493.986,A -85,B 0,C 180,E1 -12345.233,E2 -12345.233} C_VEL
LIN {X 0,Y 378.617,Z 483.626,A -85,B 0,C 180,E1 -12346.167,E2 -12346.167} C_VEL
LIN {X 0,Y 379.422,Z 471.312,A -85,B 0,C 180,E1 -12347.031,E2 -12347.031} C_VEL
LIN {X 0,Y 380.263,Z 457.855,A -85,B 0,C 180,E1 -12347.72,E2 -12347.72} C_VEL
LIN {X 0,Y 380.766,Z 445.479,A -85,B 0,C 180,E1 -12348.148,E2 -12348.148} C_VEL
LIN {X 0,Y 382.087,Z 370.655,A -85,B 0,C 180,E1 -12349.758,E2 -12349.758} C_VEL
LIN {X 0,Y 377.833,Z 337.624,A -85,B 0,C 180,E1 -12350.728,E2 -12350.728} C_VEL
LIN {X 0,Y 379.42,Z 317.732,A -85,B 0,C 180,E1 -12354.819,E2 -12354.819} C_VEL
LIN {X 0,Y 379.775,Z 313.117,A -85,B 0,C 180,E1 -12355.777,E2 -12355.777} C_VEL
LIN {X 0,Y 377.699,Z 301.761,A -85,B 0,C 180,E1 -12358.325,E2 -12358.325} C_VEL
LIN {X 0,Y 375.981,Z 293.653,A -85,B 0,C 180,E1 -12360.232,E2 -12360.232} C_VEL
LIN {X 0,Y 375.953,Z 293.655,A -85,B 0,C 180,E1 -12364.11,E2 -12364.11} C_VEL
LIN {X 0,Y 375.942,Z 293.659,A -85,B 0,C 180,E1 -12366.74,E2 -12366.74} C_VEL
LIN {X 0,Y 375.93,Z 293.654,A -85,B 0,C 180,E1 -12369.959,E2 -12369.959} C_VEL
LIN {X 0,Y 375.914,Z 293.656,A -85,B 0,C 180,E1 -12373.765,E2 -12373.765} C_VEL
LIN {X 0,Y 375.921,Z 293.661,A -85,B 0,C 180,E1 -12376.809,E2 -12376.809} C_VEL
LIN {X 0,Y 375.92,Z 293.658,A -85,B 0,C 180,E1 -12380.531,E2 -12380.531} C_VEL
LIN {X 0,Y 375.941,Z 293.655,A -85,B 0,C 180,E1 -12383.495,E2 -12383.495} C_VEL
LIN {X 0,Y 375.94,Z 293.653,A -85,B 0,C 180,E1 -12385.886,E2 -12385.886} C_VEL
LIN {X 0,Y 375.943,Z 293.654,A -85,B 0,C 180,E1 -12389.685,E2 -12389.685} C_VEL
LIN {X 0,Y 375.944,Z 293.653,A -85,B 0,C 180,E1 -12392.137,E2 -12392.137} C_VEL
LIN {X 0,Y 375.947,Z 293.654,A -85,B 0,C 180,E1 -12395.715,E2 -12395.715} C_VEL
LIN {X 0,Y 375.935,Z 293.658,A -85,B 0,C 180,E1 -12399.194,E2 -12399.194} C_VEL
LIN {X 0,Y 376.009,Z 293.646,A -85,B 0,C 180,E1 -12402.599,E2 -12402.599} C_VEL
LIN {X 0,Y 376.065,Z 293.638,A -85,B 0,C 180,E1 -12406.342,E2 -12406.342} C_VEL
LIN {X 0,Y 376.092,Z 293.635,A -85,B 0,C 180,E1 -12410.317,E2 -12410.317} C_VEL
LIN {X 0,Y 376.209,Z 293.623,A -85,B 0,C 180,E1 -12413.564,E2 -12413.564} C_VEL
LIN {X 0,Y 376.319,Z 293.609,A -85,B 0,C 180,E1 -12417.859,E2 -12417.859} C_VEL
LIN {X 0,Y 376.456,Z 293.591,A -85,B 0,C 180,E1 -12419.999,E2 -12419.999} C_VEL
LIN {X 0,Y 376.151,Z 293.632,A -85,B 0,C 180,E1 -12423.213,E2 -12423.213} C_VEL
LIN {X 0,Y 376.186,Z 293.623,A -85,B 0,C 180,E1 -12426.696,E2 -12426.696} C_VEL
LIN {X 0,Y 376.093,Z 293.638,A -85,B 0,C 180,E1 -12429.682,E2 -12429.682} C_VEL
LIN {X 0,Y 376.064,Z 293.642,A -85,B 0,C 180,E1 -12433.658,E2 -12433.658} C_VEL
LIN {X 0,Y 376.006,Z 293.65,A -85,B 0,C 180,E1 -12437.401,E2 -12437.401} C_VEL
LIN {X 0,Y 375.955,Z 293.652,A -85,B 0,C 180,E1 -12440.833,E2 -12440.833} C_VEL
LIN {X 0,Y 375.966,Z 293.653,A -85,B 0,C 180,E1 -12444.283,E2 -12444.283} C_VEL
LIN {X 0,Y 375.997,Z 293.647,A -85,B 0,C 180,E1 -12446.653,E2 -12446.653} C_VEL
LIN {X 0,Y 375.951,Z 293.653,A -85,B 0,C 180,E1 -12449.08,E2 -12449.08} C_VEL
LIN {X 0,Y 375.929,Z 293.656,A -85,B 0,C 180,E1 -12452.83,E2 -12452.83} C_VEL
LIN {X 0,Y 375.938,Z 293.656,A -85,B 0,C 180,E1 -12455.417,E2 -12455.417} C_VEL
LIN {X 0,Y 375.959,Z 293.655,A -85,B 0,C 180,E1 -12458.272,E2 -12458.272} C_VEL
LIN {X 0,Y 375.932,Z 293.658,A -85,B 0,C 180,E1 -12461.604,E2 -12461.604} C_VEL
LIN {X 0,Y 375.961,Z 293.652,A -85,B 0,C 180,E1 -12465.263,E2 -12465.263} C_VEL
LIN {X 0,Y 375.977,Z 293.653,A -85,B 0,C 180,E1 -12468.391,E2 -12468.391} C_VEL
LIN {X 0,Y 375.957,Z 293.655,A -85,B 0,C 180,E1 -12471.913,E2 -12471.913} C_VEL
LIN {X 0,Y 375.97,Z 293.651,A -85,B 0,C 180,E1 -12475.334,E2 -12475.334} C_VEL
LIN {X 0,Y 375.949,Z 293.657,A -85,B 0,C 180,E1 -12478.439,E2 -12478.439} C_VEL
LIN {X 0,Y 375.976,Z 293.652,A -85,B 0,C 180,E1 -12482.141,E2 -12482.141} C_VEL
LIN {X 0,Y 376.001,Z 293.651,A -85,B 0,C 180,E1 -12484.539,E2 -12484.539} C_VEL
LIN {X 0,Y 375.958,Z 293.654,A -85,B 0,C 180,E1 -12488.046,E2 -12488.046} C_VEL
LIN {X 0,Y 376.02,Z 293.644,A -85,B 0,C 180,E1 -12491.474,E2 -12491.474} C_VEL
LIN {X 0,Y 376.055,Z 293.642,A -85,B 0,C 180,E1 -12494.832,E2 -12494.832} C_VEL
LIN {X 0,Y 376.048,Z 293.643,A -85,B 0,C 180,E1 -12498.136,E2 -12498.136} C_VEL
LIN {X 0,Y 376.256,Z 293.615,A -85,B 0,C 180,E1 -12501.876,E2 -12501.876} C_VEL
LIN {X 0,Y 376.169,Z 293.63,A -85,B 0,C 180,E1 -12504.639,E2 -12504.639} C_VEL
LIN {X 0,Y 376.351,Z 293.603,A -85,B 0,C 180,E1 -12507.858,E2 -12507.858} C_VEL
LIN {X 0,Y 376.486,Z 293.587,A -85,B 0,C 180,E1 -12509.998,E2 -12509.998} C_VEL
LIN {X 0,Y 376.186,Z 293.625,A -85,B 0,C 180,E1 -12513.211,E2 -12513.211} C_VEL
LIN {X 0,Y 376.239,Z 293.619,A -85,B 0,C 180,E1 -12516.433,E2 -12516.433} C_VEL
LIN {X 0,Y 376.2,Z 293.624,A -85,B 0,C 180,E1 -12518.593,E2 -12518.593} C_VEL
LIN {X 0,Y 376.051,Z 293.639,A -85,B 0,C 180,E1 -12521.86,E2 -12521.86} C_VEL
LIN {X 0,Y 376.051,Z 293.643,A -85,B 0,C 180,E1 -12525.164,E2 -12525.164} C_VEL
LIN {X 0,Y 376.021,Z 293.645,A -85,B 0,C 180,E1 -12528.522,E2 -12528.522} C_VEL
LIN {X 0,Y 375.972,Z 293.649,A -85,B 0,C 180,E1 -12531.95,E2 -12531.95} C_VEL
LIN {X 0,Y 375.991,Z 293.649,A -85,B 0,C 180,E1 -12535.457,E2 -12535.457} C_VEL
LIN {X 0,Y 375.959,Z 293.657,A -85,B 0,C 180,E1 -12539.075,E2 -12539.075} C_VEL
LIN {X 0,Y 375.93,Z 293.658,A -85,B 0,C 180,E1 -12542.825,E2 -12542.825} C_VEL
LIN {X 0,Y 375.935,Z 293.657,A -85,B 0,C 180,E1 -12545.412,E2 -12545.412} C_VEL
LIN {X 0,Y 375.953,Z 293.652,A -85,B 0,C 180,E1 -12548.267,E2 -12548.267} C_VEL
LIN {X 0,Y 375.986,Z 293.652,A -85,B 0,C 180,E1 -12550.056,E2 -12550.056} C_VEL
LIN {X 0,Y 376.017,Z 294.519,A -85,B 0,C 180,E1 -12550.51,E2 -12550.51} C_VEL
LIN {X 0,Y 376.121,Z 297.239,A -85,B 0,C 180,E1 -12550.978,E2 -12550.978} C_VEL
LIN {X 0,Y 376.243,Z 301.474,A -85,B 0,C 180,E1 -12551.351,E2 -12551.351} C_VEL
LIN {X 0,Y 376.369,Z 305.405,A -85,B 0,C 180,E1 -12551.524,E2 -12551.524} C_VEL
LIN {X 0,Y 377.553,Z 313.996,A -85,B 0,C 180,E1 -12551.776,E2 -12551.776} C_VEL
LIN {X 0,Y 375.904,Z 322.653,A -85,B 0,C 180,E1 -12551.902,E2 -12551.902} C_VEL
LIN {X 0,Y 374.102,Z 405.479,A -85,B 0,C 180,E1 -12553.728,E2 -12553.728} C_VEL
LIN {X 0,Y 373.677,Z 419.466,A -85,B 0,C 180,E1 -12554.27,E2 -12554.27} C_VEL
LIN {X 0,Y 373.088,Z 431.786,A -85,B 0,C 180,E1 -12554.963,E2 -12554.963} C_VEL
LIN {X 0,Y 372.379,Z 444.043,A -85,B 0,C 180,E1 -12555.889,E2 -12555.889} C_VEL
LIN {X 0,Y 371.614,Z 454.68,A -85,B 0,C 180,E1 -12556.907,E2 -12556.907} C_VEL
LIN {X 0,Y 370.857,Z 464.969,A -85,B 0,C 180,E1 -12558.127,E2 -12558.127} C_VEL
LIN {X 0,Y 370.028,Z 474.87,A -85,B 0,C 180,E1 -12559.591,E2 -12559.591} C_VEL
LIN {X 0,Y 369.263,Z 484.073,A -85,B 0,C 180,E1 -12561.281,E2 -12561.281} C_VEL
LIN {X 0,Y 368.741,Z 490.909,A -85,B 0,C 180,E1 -12562.859,E2 -12562.859} C_VEL
LIN {X 0,Y 368.307,Z 496.341,A -85,B 0,C 180,E1 -12564.409,E2 -12564.409} C_VEL
LIN {X 0,Y 367.95,Z 501.626,A -85,B 0,C 180,E1 -12566.365,E2 -12566.365} C_VEL
LIN {X 0,Y 367.735,Z 504.257,A -85,B 0,C 180,E1 -12567.648,E2 -12567.648} C_VEL
LIN {X 0,Y 367.494,Z 506.806,A -85,B 0,C 180,E1 -12569.369,E2 -12569.369} C_VEL
LIN {X 0,Y 367.441,Z 508.474,A -85,B 0,C 180,E1 -12571.435,E2 -12571.435} C_VEL
LIN {X 0,Y 367.425,Z 508.79,A -85,B 0,C 180,E1 -12572.674,E2 -12572.674} C_VEL
LIN {X 0,Y 367.508,Z 508.511,A -85,B 0,C 180,E1 -12573.985,E2 -12573.985} C_VEL
LIN {X 0,Y 367.651,Z 507.82,A -85,B 0,C 180,E1 -12575.131,E2 -12575.131} C_VEL
LIN {X 0,Y 367.861,Z 506.372,A -85,B 0,C 180,E1 -12576.479,E2 -12576.479} C_VEL
LIN {X 0,Y 368.217,Z 503.699,A -85,B 0,C 180,E1 -12578.15,E2 -12578.15} C_VEL
LIN {X 0,Y 368.653,Z 499.676,A -85,B 0,C 180,E1 -12579.932,E2 -12579.932} C_VEL
LIN {X 0,Y 369.272,Z 494.623,A -85,B 0,C 180,E1 -12581.618,E2 -12581.618} C_VEL
LIN {X 0,Y 370.03,Z 488.778,A -85,B 0,C 180,E1 -12583.164,E2 -12583.164} C_VEL
LIN {X 0,Y 370.843,Z 482.049,A -85,B 0,C 180,E1 -12584.615,E2 -12584.615} C_VEL
LIN {X 0,Y 371.814,Z 473.861,A -85,B 0,C 180,E1 -12586.055,E2 -12586.055} C_VEL
LIN {X 0,Y 372.927,Z 463.81,A -85,B 0,C 180,E1 -12587.484,E2 -12587.484} C_VEL
LIN {X 0,Y 374.004,Z 453.652,A -85,B 0,C 180,E1 -12588.647,E2 -12588.647} C_VEL
LIN {X 0,Y 374.891,Z 443.322,A -85,B 0,C 180,E1 -12589.605,E2 -12589.605} C_VEL
LIN {X 0,Y 375.769,Z 431.509,A -85,B 0,C 180,E1 -12590.459,E2 -12590.459} C_VEL
LIN {X 0,Y 376.444,Z 418.43,A -85,B 0,C 180,E1 -12591.168,E2 -12591.168} C_VEL
LIN {X 0,Y 376.998,Z 404.802,A -85,B 0,C 180,E1 -12591.652,E2 -12591.652} C_VEL
LIN {X 0,Y 379.358,Z 320.482,A -85,B 0,C 180,E1 -12593.619,E2 -12593.619} C_VEL
LIN {X 0,Y 377.207,Z 314.245,A -85,B 0,C 180,E1 -12593.952,E2 -12593.952} C_VEL
LIN {X 0,Y 371.918,Z 302.129,A -85,B 0,C 180,E1 -12594.715,E2 -12594.715} C_VEL
LIN {X 0,Y 370.229,Z 298.8,A -85,B 0,C 180,E1 -12594.964,E2 -12594.964} C_VEL
LIN {X 0,Y 368.976,Z 294.531,A -85,B 0,C 180,E1 -12596.007,E2 -12596.007} C_VEL
LIN {X 0,Y 369.268,Z 294.492,A -85,B 0,C 180,E1 -12597.819,E2 -12597.819} C_VEL
LIN {X 0,Y 369.407,Z 294.47,A -85,B 0,C 180,E1 -12600.001,E2 -12600.001} C_VEL
LIN {X 0,Y 369.268,Z 294.488,A -85,B 0,C 180,E1 -12602.182,E2 -12602.182} C_VEL
LIN {X 0,Y 369.149,Z 294.501,A -85,B 0,C 180,E1 -12606.56,E2 -12606.56} C_VEL
LIN {X 0,Y 369.021,Z 294.516,A -85,B 0,C 180,E1 -12609.87,E2 -12609.87} C_VEL
LIN {X 0,Y 368.992,Z 294.521,A -85,B 0,C 180,E1 -12613.774,E2 -12613.774} C_VEL
LIN {X 0,Y 368.947,Z 294.522,A -85,B 0,C 180,E1 -12617.745,E2 -12617.745} C_VEL
LIN {X 0,Y 368.867,Z 294.536,A -85,B 0,C 180,E1 -12621.224,E2 -12621.224} C_VEL
LIN {X 0,Y 368.914,Z 294.532,A -85,B 0,C 180,E1 -12624.779,E2 -12624.779} C_VEL
LIN {X 0,Y 368.923,Z 294.533,A -85,B 0,C 180,E1 -12627.207,E2 -12627.207} C_VEL
LIN {X 0,Y 368.875,Z 294.535,A -85,B 0,C 180,E1 -12630.991,E2 -12630.991} C_VEL
LIN {X 0,Y 368.902,Z 294.528,A -85,B 0,C 180,E1 -12634.858,E2 -12634.858} C_VEL
LIN {X 0,Y 368.881,Z 294.535,A -85,B 0,C 180,E1 -12638.645,E2 -12638.645} C_VEL
LIN {X 0,Y 368.866,Z 294.533,A -85,B 0,C 180,E1 -12641.825,E2 -12641.825} C_VEL
LIN {X 0,Y 368.853,Z 294.539,A -85,B 0,C 180,E1 -12645.18,E2 -12645.18} C_VEL
LIN {X 0,Y 368.859,Z 294.538,A -85,B 0,C 180,E1 -12648.182,E2 -12648.182} C_VEL
LIN {X 0,Y 368.884,Z 294.538,A -85,B 0,C 180,E1 -12651.365,E2 -12651.365} C_VEL
LIN {X 0,Y 368.919,Z 294.535,A -85,B 0,C 180,E1 -12655.151,E2 -12655.151} C_VEL
LIN {X 0,Y 368.9,Z 294.576,A -85,B 0,C 180,E1 -12658.863,E2 -12658.863} C_VEL
LIN {X 0,Y 371.739,Z 305.697,A -85,B 0,C 180,E1 -12661.53,E2 -12661.53} C_VEL
LIN {X 0,Y 373.581,Z 315.692,A -85,B 0,C 180,E1 -12663.767,E2 -12663.767} C_VEL
LIN {X 0,Y 372.139,Z 333.54,A -85,B 0,C 180,E1 -12667.277,E2 -12667.277} C_VEL
LIN {X 0,Y 375.907,Z 353.879,A -85,B 0,C 180,E1 -12668.109,E2 -12668.109} C_VEL
LIN {X 0,Y 377.921,Z 369.35,A -85,B 0,C 180,E1 -12668.659,E2 -12668.659} C_VEL
LIN {X 0,Y 378.251,Z 374.399,A -85,B 0,C 180,E1 -12668.812,E2 -12668.812} C_VEL
LIN {X 0,Y 376.275,Z 445.515,A -85,B 0,C 180,E1 -12670.465,E2 -12670.465} C_VEL
LIN {X 0,Y 375.466,Z 458.323,A -85,B 0,C 180,E1 -12670.954,E2 -12670.954} C_VEL
LIN {X 0,Y 374.417,Z 471.41,A -85,B 0,C 180,E1 -12671.679,E2 -12671.679} C_VEL
LIN {X 0,Y 373.27,Z 483.814,A -85,B 0,C 180,E1 -12672.612,E2 -12672.612} C_VEL
LIN {X 0,Y 372.135,Z 495.026,A -85,B 0,C 180,E1 -12673.688,E2 -12673.688} C_VEL
LIN {X 0,Y 371.009,Z 504.976,A -85,B 0,C 180,E1 -12674.875,E2 -12674.875} C_VEL
LIN {X 0,Y 370.012,Z 514.45,A -85,B 0,C 180,E1 -12676.269,E2 -12676.269} C_VEL
LIN {X 0,Y 369.089,Z 523.545,A -85,B 0,C 180,E1 -12677.913,E2 -12677.913} C_VEL
LIN {X 0,Y 368.32,Z 530.874,A -85,B 0,C 180,E1 -12679.559,E2 -12679.559} C_VEL
LIN {X 0,Y 367.871,Z 536.751,A -85,B 0,C 180,E1 -12681.211,E2 -12681.211} C_VEL
LIN {X 0,Y 367.625,Z 541.398,A -85,B 0,C 180,E1 -12682.864,E2 -12682.864} C_VEL
LIN {X 0,Y 367.478,Z 544.932,A -85,B 0,C 180,E1 -12684.515,E2 -12684.515} C_VEL
LIN {X 0,Y 367.503,Z 546.709,A -85,B 0,C 180,E1 -12685.615,E2 -12685.615} C_VEL
LIN {X 0,Y 367.448,Z 548.065,A -85,B 0,C 180,E1 -12686.713,E2 -12686.713} C_VEL
LIN {X 0,Y 367.529,Z 548.986,A -85,B 0,C 180,E1 -12687.81,E2 -12687.81} C_VEL
LIN {X 0,Y 367.587,Z 549.461,A -85,B 0,C 180,E1 -12688.906,E2 -12688.906} C_VEL
LIN {X 0,Y 367.59,Z 549.526,A -85,B 0,C 180,E1 -12690.002,E2 -12690.002} C_VEL
LIN {X 0,Y 367.598,Z 549.184,A -85,B 0,C 180,E1 -12691.097,E2 -12691.097} C_VEL
LIN {X 0,Y 367.601,Z 548.389,A -85,B 0,C 180,E1 -12692.193,E2 -12692.193} C_VEL
LIN {X 0,Y 367.483,Z 547.143,A -85,B 0,C 180,E1 -12693.291,E2 -12693.291} C_VEL
LIN {X 0,Y 367.569,Z 544.464,A -85,B 0,C 180,E1 -12694.937,E2 -12694.937} C_VEL
LIN {X 0,Y 367.638,Z 540.698,A -85,B 0,C 180,E1 -12696.587,E2 -12696.587} C_VEL
LIN {X 0,Y 367.775,Z 535.75,A -85,B 0,C 180,E1 -12698.241,E2 -12698.241} C_VEL
LIN {X 0,Y 368.102,Z 529.48,A -85,B 0,C 180,E1 -12699.895,E2 -12699.895} C_VEL
LIN {X 0,Y 368.657,Z 521.651,A -85,B 0,C 180,E1 -12701.547,E2 -12701.547} C_VEL
LIN {X 0,Y 369.252,Z 513.602,A -85,B 0,C 180,E1 -12702.923,E2 -12702.923} C_VEL
LIN {X 0,Y 370.064,Z 503.784,A -85,B 0,C 180,E1 -12704.294,E2 -12704.294} C_VEL
LIN {X 0,Y 370.897,Z 492.889,A -85,B 0,C 180,E1 -12705.525,E2 -12705.525} C_VEL
LIN {X 0,Y 371.726,Z 482.325,A -85,B 0,C 180,E1 -12706.475,E2 -12706.475} C_VEL
LIN {X 0,Y 372.578,Z 469.711,A -85,B 0,C 180,E1 -12707.354,E2 -12707.354} C_VEL
LIN {X 0,Y 373.435,Z 456.609,A -85,B 0,C 180,E1 -12708.02,E2 -12708.02} C_VEL
LIN {X 0,Y 373.93,Z 443.551,A -85,B 0,C 180,E1 -12708.456,E2 -12708.456} C_VEL
LIN {X 0,Y 375.298,Z 371.627,A -85,B 0,C 180,E1 -12710.034,E2 -12710.034} C_VEL
LIN {X 0,Y 370.925,Z 337.293,A -85,B 0,C 180,E1 -12711.058,E2 -12711.058} C_VEL
LIN {X 0,Y 372.643,Z 316.929,A -85,B 0,C 180,E1 -12715.323,E2 -12715.323} C_VEL
LIN {X 0,Y 372.77,Z 313.778,A -85,B 0,C 180,E1 -12715.997,E2 -12715.997} C_VEL
LIN {X 0,Y 370.493,Z 301.997,A -85,B 0,C 180,E1 -12718.709,E2 -12718.709} C_VEL
LIN {X 0,Y 368.919,Z 294.533,A -85,B 0,C 180,E1 -12720.477,E2 -12720.477} C_VEL
LIN {X 0,Y 368.891,Z 294.532,A -85,B 0,C 180,E1 -12723.537,E2 -12723.537} C_VEL
LIN {X 0,Y 368.889,Z 294.536,A -85,B 0,C 180,E1 -12726.852,E2 -12726.852} C_VEL
LIN {X 0,Y 368.876,Z 294.535,A -85,B 0,C 180,E1 -12730.372,E2 -12730.372} C_VEL
LIN {X 0,Y 368.868,Z 294.534,A -85,B 0,C 180,E1 -12733.613,E2 -12733.613} C_VEL
LIN {X 0,Y 368.872,Z 294.538,A -85,B 0,C 180,E1 -12736.693,E2 -12736.693} C_VEL
LIN {X 0,Y 368.872,Z 294.534,A -85,B 0,C 180,E1 -12739.646,E2 -12739.646} C_VEL
LIN {X 0,Y 368.88,Z 294.536,A -85,B 0,C 180,E1 -12743.144,E2 -12743.144} C_VEL
LIN {X 0,Y 368.878,Z 294.534,A -85,B 0,C 180,E1 -12746.459,E2 -12746.459} C_VEL
LIN {X 0,Y 368.882,Z 294.533,A -85,B 0,C 180,E1 -12750.306,E2 -12750.306} C_VEL
LIN {X 0,Y 368.911,Z 294.529,A -85,B 0,C 180,E1 -12754.013,E2 -12754.013} C_VEL
LIN {X 0,Y 368.876,Z 294.536,A -85,B 0,C 180,E1 -12757.601,E2 -12757.601} C_VEL
LIN {X 0,Y 368.924,Z 294.533,A -85,B 0,C 180,E1 -12761.104,E2 -12761.104} C_VEL
LIN {X 0,Y 368.971,Z 294.522,A -85,B 0,C 180,E1 -12764.533,E2 -12764.533} C_VEL
LIN {X 0,Y 368.979,Z 294.522,A -85,B 0,C 180,E1 -12767.905,E2 -12767.905} C_VEL
LIN {X 0,Y 369.14,Z 294.503,A -85,B 0,C 180,E1 -12771.87,E2 -12771.87} C_VEL
LIN {X 0,Y 369.11,Z 294.505,A -85,B 0,C 180,E1 -12774.537,E2 -12774.537} C_VEL
LIN {X 0,Y 369.285,Z 294.486,A -85,B 0,C 180,E1 -12777.818,E2 -12777.818} C_VEL
LIN {X 0,Y 369.405,Z 294.469,A -85,B 0,C 180,E1 -12779.999,E2 -12779.999} C_VEL
LIN {X 0,Y 369.284,Z 294.484,A -85,B 0,C 180,E1 -12782.181,E2 -12782.181} C_VEL
LIN {X 0,Y 369.156,Z 294.499,A -85,B 0,C 180,E1 -12786.682,E2 -12786.682} C_VEL
LIN {X 0,Y 369.042,Z 294.517,A -85,B 0,C 180,E1 -12789.868,E2 -12789.868} C_VEL
LIN {X 0,Y 369.012,Z 294.52,A -85,B 0,C 180,E1 -12793.772,E2 -12793.772} C_VEL
LIN {X 0,Y 368.967,Z 294.526,A -85,B 0,C 180,E1 -12797.743,E2 -12797.743} C_VEL
LIN {X 0,Y 368.886,Z 294.534,A -85,B 0,C 180,E1 -12801.222,E2 -12801.222} C_VEL
LIN {X 0,Y 368.932,Z 294.527,A -85,B 0,C 180,E1 -12804.777,E2 -12804.777} C_VEL
LIN {X 0,Y 368.946,Z 294.526,A -85,B 0,C 180,E1 -12807.204,E2 -12807.204} C_VEL
LIN {X 0,Y 368.899,Z 294.535,A -85,B 0,C 180,E1 -12809.691,E2 -12809.691} C_VEL
LIN {X 0,Y 368.877,Z 294.534,A -85,B 0,C 180,E1 -12813.044,E2 -12813.044} C_VEL
LIN {X 0,Y 368.899,Z 294.535,A -85,B 0,C 180,E1 -12816.198,E2 -12816.198} C_VEL
LIN {X 0,Y 368.889,Z 294.532,A -85,B 0,C 180,E1 -12818.954,E2 -12818.954} C_VEL
LIN {X 0,Y 368.875,Z 294.538,A -85,B 0,C 180,E1 -12822.012,E2 -12822.012} C_VEL
LIN {X 0,Y 368.936,Z 294.527,A -85,B 0,C 180,E1 -12825.188,E2 -12825.188} C_VEL
LIN {X 0,Y 368.928,Z 294.531,A -85,B 0,C 180,E1 -12828.187,E2 -12828.187} C_VEL
LIN {X 0,Y 368.901,Z 294.531,A -85,B 0,C 180,E1 -12831.36,E2 -12831.36} C_VEL
LIN {X 0,Y 368.927,Z 294.528,A -85,B 0,C 180,E1 -12835.147,E2 -12835.147} C_VEL
LIN {X 0,Y 368.922,Z 294.528,A -85,B 0,C 180,E1 -12839.047,E2 -12839.047} C_VEL
LIN {X 0,Y 368.957,Z 294.526,A -85,B 0,C 180,E1 -12842.797,E2 -12842.797} C_VEL
LIN {X 0,Y 368.94,Z 294.529,A -85,B 0,C 180,E1 -12846.113,E2 -12846.113} C_VEL
LIN {X 0,Y 368.933,Z 294.529,A -85,B 0,C 180,E1 -12849.947,E2 -12849.947} C_VEL
LIN {X 0,Y 368.972,Z 294.522,A -85,B 0,C 180,E1 -12853.398,E2 -12853.398} C_VEL
LIN {X 0,Y 369.055,Z 294.515,A -85,B 0,C 180,E1 -12856.79,E2 -12856.79} C_VEL
LIN {X 0,Y 369.065,Z 294.513,A -85,B 0,C 180,E1 -12860.131,E2 -12860.131} C_VEL
LIN {X 0,Y 369.186,Z 294.498,A -85,B 0,C 180,E1 -12862.341,E2 -12862.341} C_VEL
LIN {X 0,Y 369.142,Z 294.505,A -85,B 0,C 180,E1 -12864.536,E2 -12864.536} C_VEL
LIN {X 0,Y 369.316,Z 294.479,A -85,B 0,C 180,E1 -12867.817,E2 -12867.817} C_VEL
LIN {X 0,Y 369.456,Z 294.462,A -85,B 0,C 180,E1 -12869.998,E2 -12869.998} C_VEL
LIN {X 0,Y 369.316,Z 294.48,A -85,B 0,C 180,E1 -12872.179,E2 -12872.179} C_VEL
LIN {X 0,Y 369.201,Z 294.496,A -85,B 0,C 180,E1 -12876.556,E2 -12876.556} C_VEL
LIN {X 0,Y 369.133,Z 294.506,A -85,B 0,C 180,E1 -12878.758,E2 -12878.758} C_VEL
LIN {X 0,Y 369.006,Z 294.518,A -85,B 0,C 180,E1 -12882.09,E2 -12882.09} C_VEL
LIN {X 0,Y 368.99,Z 294.52,A -85,B 0,C 180,E1 -12885.462,E2 -12885.462} C_VEL
LIN {X 0,Y 368.982,Z 294.525,A -85,B 0,C 180,E1 -12888.889,E2 -12888.889} C_VEL
